gfCNCPoint3[20419] = {X 583.3023, Y 48.9046, Z -4.6667, A 0.000, B 0.000, C 0.000 }
gfCNCPoint3[20420] = {X 582.3585, Y 49.2242, Z -4.6667, A 0.000, B 0.000, C 0.000 }
gfCNCPoint3[20421] = {X 581.3666, Y 49.3191, Z -4.6667, A 0.000, B 0.000, C 0.000 }
gfCNCPoint3[20422] = {X 580.3794, Y 49.1842, Z -4.6667, A 0.000, B 0.000, C 0.000 }
gfCNCPoint3[20423] = {X 579.4493, Y 48.8268, Z -4.6667, A 0.000, B 0.000, C 0.000 }
gfCNCPoint3[20424] = {X 578.6259, Y 48.2657, Z -4.6667, A 0.000, B 0.000, C 0.000 }
gfCNCPoint3[20425] = {X 577.9529, Y 47.5309, Z -4.6667, A 0.000, B 0.000, C 0.000 }
gfCNCPoint3[20426] = {X 577.4662, Y 46.6615, Z -4.6667, A 0.000, B 0.000, C 0.000 }
gfCNCPoint3[20427] = {X 572.0189, Y 33.3415, Z -4.6667, A 0.000, B 0.000, C 0.000 }
gfCNCPoint3[20428] = {X 572.0192, Y 40.7711, Z -4.6667, A 0.000, B 0.000, C 0.000 }
gfCNCPoint3[20429] = {X 572.6574, Y 41.4420, Z -4.6667, A 0.000, B 0.000, C 0.000 }
gfCNCPoint3[20430] = {X 573.1380, Y 42.2334, Z -4.6667, A 0.000, B 0.000, C 0.000 }
gfCNCPoint3[20431] = {X 573.4389, Y 43.1090, Z -4.6667, A 0.000, B 0.000, C 0.000 }
gfCNCPoint3[20432] = {X 573.5463, Y 44.0287, Z -4.6667, A 0.000, B 0.000, C 0.000 }
gfCNCPoint3[20433] = {X 573.5464, Y 45.0000, Z -4.6667, A 0.000, B 0.000, C 0.000 }
gfCNCPoint3[20434] = {X 573.4381, Y 45.9613, Z -4.6667, A 0.000, B 0.000, C 0.000 }
gfCNCPoint3[20435] = {X 573.1186, Y 46.8744, Z -4.6667, A 0.000, B 0.000, C 0.000 }
gfCNCPoint3[20436] = {X 572.6039, Y 47.6935, Z -4.6667, A 0.000, B 0.000, C 0.000 }
gfCNCPoint3[20437] = {X 571.9199, Y 48.3775, Z -4.6667, A 0.000, B 0.000, C 0.000 }
gfCNCPoint3[20438] = {X 571.1008, Y 48.8922, Z -4.6667, A 0.000, B 0.000, C 0.000 }
gfCNCPoint3[20439] = {X 570.1877, Y 49.2117, Z -4.6667, A 0.000, B 0.000, C 0.000 }
gfCNCPoint3[20440] = {X 569.2264, Y 49.3200, Z -4.6667, A 0.000, B 0.000, C 0.000 }
gfCNCPoint3[20441] = {X 562.4443, Y 49.3200, Z -4.6667, A 0.000, B 0.000, C 0.000 }
gfCNCPoint3[20442] = {X 561.4830, Y 49.2117, Z -4.6667, A 0.000, B 0.000, C 0.000 }
gfCNCPoint3[20443] = {X 560.5699, Y 48.8922, Z -4.6667, A 0.000, B 0.000, C 0.000 }
gfCNCPoint3[20444] = {X 559.7508, Y 48.3775, Z -4.6667, A 0.000, B 0.000, C 0.000 }
gfCNCPoint3[20445] = {X 559.0668, Y 47.6935, Z -4.6667, A 0.000, B 0.000, C 0.000 }
gfCNCPoint3[20446] = {X 558.5521, Y 46.8744, Z -4.6667, A 0.000, B 0.000, C 0.000 }
gfCNCPoint3[20447] = {X 558.2326, Y 45.9613, Z -4.6667, A 0.000, B 0.000, C 0.000 }
gfCNCPoint3[20448] = {X 558.1243, Y 45.0000, Z -4.6667, A 0.000, B 0.000, C 0.000 }
gfCNCPoint3[20449] = {X 558.1243, Y 44.0647, Z -4.6667, A 0.000, B 0.000, C 0.000 }
gfCNCPoint3[20450] = {X 558.2284, Y 43.1360, Z -4.6667, A 0.000, B 0.000, C 0.000 }
gfCNCPoint3[20451] = {X 558.5283, Y 42.2510, Z -4.6667, A 0.000, B 0.000, C 0.000 }
gfCNCPoint3[20452] = {X 559.0102, Y 41.4503, Z -4.6667, A 0.000, B 0.000, C 0.000 }
gfCNCPoint3[20453] = {X 559.6518, Y 40.7709, Z -4.6667, A 0.000, B 0.000, C 0.000 }
gfCNCPoint3[20454] = {X 559.6518, Y 9.2302, Z -4.6667, A 0.000, B 0.000, C 0.000 }
gfCNCPoint3[20455] = {X 559.0134, Y 8.5592, Z -4.6667, A 0.000, B 0.000, C 0.000 }
gfCNCPoint3[20456] = {X 558.5327, Y 7.7676, Z -4.6667, A 0.000, B 0.000, C 0.000 }
gfCNCPoint3[20457] = {X 558.2318, Y 6.8917, Z -4.6667, A 0.000, B 0.000, C 0.000 }
gfCNCPoint3[20458] = {X 558.1245, Y 5.9718, Z -4.6667, A 0.000, B 0.000, C 0.000 }
gfCNCPoint3[20459] = {X 558.1243, Y 5.0000, Z -4.6667, A 0.000, B 0.000, C 0.000 }
gfCNCPoint3[20460] = {X 558.2326, Y 4.0387, Z -4.6667, A 0.000, B 0.000, C 0.000 }
gfCNCPoint3[20461] = {X 558.5521, Y 3.1256, Z -4.6667, A 0.000, B 0.000, C 0.000 }
gfCNCPoint3[20462] = {X 559.0668, Y 2.3065, Z -4.6667, A 0.000, B 0.000, C 0.000 }
gfCNCPoint3[20463] = {X 559.7508, Y 1.6225, Z -4.6667, A 0.000, B 0.000, C 0.000 }
gfCNCPoint3[20464] = {X 560.5699, Y 1.1078, Z -4.6667, A 0.000, B 0.000, C 0.000 }
gfCNCPoint3[20465] = {X 561.4830, Y 0.7883, Z -4.6667, A 0.000, B 0.000, C 0.000 }
gfCNCPoint3[20466] = {X 562.4443, Y 0.6800, Z -4.6667, A 0.000, B 0.000, C 0.000 }
gfCNCPoint3[20467] = {X 570.9376, Y 0.6800, Z -4.6667, A 0.000, B 0.000, C 0.000 }
gfCNCPoint3[20468] = {X 571.8988, Y 0.7883, Z -4.6667, A 0.000, B 0.000, C 0.000 }
gfCNCPoint3[20469] = {X 572.8119, Y 1.1078, Z -4.6667, A 0.000, B 0.000, C 0.000 }
gfCNCPoint3[20470] = {X 573.6310, Y 1.6225, Z -4.6667, A 0.000, B 0.000, C 0.000 }
gfCNCPoint3[20471] = {X 574.3151, Y 2.3065, Z -4.6667, A 0.000, B 0.000, C 0.000 }
gfCNCPoint3[20472] = {X 574.8297, Y 3.1256, Z -4.6667, A 0.000, B 0.000, C 0.000 }
gfCNCPoint3[20473] = {X 575.1492, Y 4.0387, Z -4.6667, A 0.000, B 0.000, C 0.000 }
gfCNCPoint3[20474] = {X 575.2576, Y 5.0000, Z -4.6667, A 0.000, B 0.000, C 0.000 }
gfCNCPoint3[20475] = {X 575.2576, Y 5.9342, Z -4.6667, A 0.000, B 0.000, C 0.000 }
gfCNCPoint3[20476] = {X 575.1835, Y 6.7305, Z -4.6667, A 0.000, B 0.000, C 0.000 }
gfCNCPoint3[20477] = {X 574.9639, Y 7.4995, Z -4.6667, A 0.000, B 0.000, C 0.000 }
gfCNCPoint3[20478] = {X 574.6064, Y 8.2149, Z -4.6667, A 0.000, B 0.000, C 0.000 }
gfCNCPoint3[20479] = {X 581.1910, Y 24.3698, Z -4.6667, A 0.000, B 0.000, C 0.000 }
gfCNCPoint3[20480] = {X 587.8458, Y 8.0941, Z -4.6667, A 0.000, B 0.000, C 0.000 }
gfCNCPoint3[20481] = {X 587.5317, Y 7.4230, Z -4.6667, A 0.000, B 0.000, C 0.000 }
gfCNCPoint3[20482] = {X 587.3369, Y 6.7082, Z -4.6667, A 0.000, B 0.000, C 0.000 }
gfCNCPoint3[20483] = {X 587.2671, Y 5.9705, Z -4.6667, A 0.000, B 0.000, C 0.000 }
gfCNCPoint3[20484] = {X 587.2670, Y 5.0000, Z -4.6667, A 0.000, B 0.000, C 0.000 }
gfCNCPoint3[20485] = {X 587.3753, Y 4.0387, Z -4.6667, A 0.000, B 0.000, C 0.000 }
gfCNCPoint3[20486] = {X 587.6948, Y 3.1256, Z -4.6667, A 0.000, B 0.000, C 0.000 }
gfCNCPoint3[20487] = {X 588.2094, Y 2.3065, Z -4.6667, A 0.000, B 0.000, C 0.000 }
gfCNCPoint3[20488] = {X 588.8935, Y 1.6225, Z -4.6667, A 0.000, B 0.000, C 0.000 }
gfCNCPoint3[20489] = {X 589.7126, Y 1.1078, Z -4.6667, A 0.000, B 0.000, C 0.000 }
gfCNCPoint3[20490] = {X 590.6257, Y 0.7883, Z -4.6667, A 0.000, B 0.000, C 0.000 }
gfCNCPoint3[20491] = {X 591.5870, Y 0.6800, Z -4.6667, A 0.000, B 0.000, C 0.000 }
gfCNCPoint3[20492] = {X 600.0000, Y 0.6800, Z -4.6667, A 0.000, B 0.000, C 0.000 }
gfCNCPoint3[20493] = {X 600.8562, Y 0.7657, Z -4.6667, A 0.000, B 0.000, C 0.000 }
gfCNCPoint3[20494] = {X 601.6783, Y 1.0194, Z -4.6667, A 0.000, B 0.000, C 0.000 }
gfCNCPoint3[20495] = {X 602.4340, Y 1.4309, Z -4.6667, A 0.000, B 0.000, C 0.000 }
gfCNCPoint3[20496] = {X 603.0930, Y 1.9841, Z -4.6667, A 0.000, B 0.000, C 0.000 }
gfCNCPoint3[20497] = {X 603.6294, Y 2.6569, Z -4.6667, A 0.000, B 0.000, C 0.000 }
gfCNCPoint3[20498] = {X 603.6634, Y 2.7104, Z -4.6667, A 0.000, B 0.000, C 0.000 }
gfCNCPoint3[20499] = {X 603.6966, Y 2.7644, Z -4.6667, A 0.000, B 0.000, C 0.000 }
gfCNCPoint3[20500] = {X 608.0000, Y 9.8803, Z -4.6667, A 0.000, B 0.000, C 0.000 }
gfCNCPoint3[20501] = {X 608.0000, Y 9.8803, Z -1.6667, A 0.000, B 0.000, C 0.000 }
gfCNCPoint3[20502] = {X 608.0000, Y 9.8803, Z 11.0000, A 0.000, B 0.000, C 0.000 }
gfCNCPoint3[20503] = {X -7.6966, Y 16.7865, Z 11.0000, A 0.000, B 0.000, C 0.000 }
gfCNCPoint3[20504] = {X -7.6966, Y 16.7865, Z -1.6667, A 0.000, B 0.000, C 0.000 }
gfCNCPoint3[20505] = {X -7.6966, Y 16.7865, Z -4.6667, A 0.000, B 0.000, C 0.000 }
gfCNCPoint3[20506] = {X -4.6244, Y 16.7865, Z -4.6667, A 0.000, B 0.000, C 0.000 }
gfCNCPoint3[20507] = {X -3.6966, Y 12.8956, Z -4.6667, A 0.000, B 0.000, C 0.000 }
gfCNCPoint3[20508] = {X -3.6291, Y 12.6465, Z -4.6667, A 0.000, B 0.000, C 0.000 }
gfCNCPoint3[20509] = {X -3.5466, Y 12.4020, Z -4.6667, A 0.000, B 0.000, C 0.000 }
gfCNCPoint3[20510] = {X -3.1001, Y 11.5272, Z -4.6667, A 0.000, B 0.000, C 0.000 }
gfCNCPoint3[20511] = {X -2.4643, Y 10.7786, Z -4.6667, A 0.000, B 0.000, C 0.000 }
gfCNCPoint3[20512] = {X -1.6733, Y 10.1963, Z -4.6667, A 0.000, B 0.000, C 0.000 }
gfCNCPoint3[20513] = {X -1.0760, Y 9.8556, Z -4.6667, A 0.000, B 0.000, C 0.000 }
gfCNCPoint3[20514] = {X -0.1979, Y 9.4786, Z -4.6667, A 0.000, B 0.000, C 0.000 }
gfCNCPoint3[20515] = {X 0.7423, Y 9.3079, Z -4.6667, A 0.000, B 0.000, C 0.000 }
gfCNCPoint3[20516] = {X 1.6969, Y 9.3520, Z -4.6667, A 0.000, B 0.000, C 0.000 }
gfCNCPoint3[20517] = {X 2.6173, Y 9.6089, Z -4.6667, A 0.000, B 0.000, C 0.000 }
gfCNCPoint3[20518] = {X 3.4039, Y 9.2325, Z -4.6667, A 0.000, B 0.000, C 0.000 }
gfCNCPoint3[20519] = {X 4.2182, Y 8.9206, Z -4.6667, A 0.000, B 0.000, C 0.000 }
gfCNCPoint3[20520] = {X 6.1238, Y 8.2532, Z -4.6667, A 0.000, B 0.000, C 0.000 }
gfCNCPoint3[20521] = {X 8.0799, Y 7.7526, Z -4.6667, A 0.000, B 0.000, C 0.000 }
gfCNCPoint3[20522] = {X 10.0718, Y 7.4226, Z -4.6667, A 0.000, B 0.000, C 0.000 }
gfCNCPoint3[20523] = {X 12.0848, Y 7.2658, Z -4.6667, A 0.000, B 0.000, C 0.000 }
gfCNCPoint3[20524] = {X 14.1038, Y 7.2832, Z -4.6667, A 0.000, B 0.000, C 0.000 }
gfCNCPoint3[20525] = {X 16.1138, Y 7.4747, Z -4.6667, A 0.000, B 0.000, C 0.000 }
gfCNCPoint3[20526] = {X 17.9288, Y 7.8067, Z -4.6667, A 0.000, B 0.000, C 0.000 }
gfCNCPoint3[20527] = {X 19.6983, Y 8.3293, Z -4.6667, A 0.000, B 0.000, C 0.000 }
gfCNCPoint3[20528] = {X 21.4023, Y 9.0367, Z -4.6667, A 0.000, B 0.000, C 0.000 }
gfCNCPoint3[20529] = {X 23.0218, Y 9.9207, Z -4.6667, A 0.000, B 0.000, C 0.000 }
gfCNCPoint3[20530] = {X 24.5384, Y 10.9716, Z -4.6667, A 0.000, B 0.000, C 0.000 }
gfCNCPoint3[20531] = {X 25.6169, Y 11.9146, Z -4.6667, A 0.000, B 0.000, C 0.000 }
gfCNCPoint3[20532] = {X 26.5844, Y 12.9712, Z -4.6667, A 0.000, B 0.000, C 0.000 }
gfCNCPoint3[20533] = {X 27.4289, Y 14.1285, Z -4.6667, A 0.000, B 0.000, C 0.000 }
gfCNCPoint3[20534] = {X 28.1401, Y 15.3722, Z -4.6667, A 0.000, B 0.000, C 0.000 }
gfCNCPoint3[20535] = {X 28.7091, Y 16.6870, Z -4.6667, A 0.000, B 0.000, C 0.000 }
gfCNCPoint3[20536] = {X 29.1816, Y 18.3343, Z -4.6667, A 0.000, B 0.000, C 0.000 }
gfCNCPoint3[20537] = {X 29.4619, Y 20.0250, Z -4.6667, A 0.000, B 0.000, C 0.000 }
gfCNCPoint3[20538] = {X 29.5464, Y 21.7367, Z -4.6667, A 0.000, B 0.000, C 0.000 }
gfCNCPoint3[20539] = {X 29.4338, Y 23.4467, Z -4.6667, A 0.000, B 0.000, C 0.000 }
gfCNCPoint3[20540] = {X 29.1258, Y 25.1326, Z -4.6667, A 0.000, B 0.000, C 0.000 }
gfCNCPoint3[20541] = {X 28.6966, Y 26.5422, Z -4.6667, A 0.000, B 0.000, C 0.000 }
gfCNCPoint3[20542] = {X 28.0924, Y 27.8862, Z -4.6667, A 0.000, B 0.000, C 0.000 }
gfCNCPoint3[20543] = {X 27.3227, Y 29.1428, Z -4.6667, A 0.000, B 0.000, C 0.000 }
gfCNCPoint3[20544] = {X 26.4001, Y 30.2918, Z -4.6667, A 0.000, B 0.000, C 0.000 }
gfCNCPoint3[20545] = {X 25.3394, Y 31.3146, Z -4.6667, A 0.000, B 0.000, C 0.000 }
gfCNCPoint3[20546] = {X 25.2268, Y 31.4090, Z -4.6667, A 0.000, B 0.000, C 0.000 }
gfCNCPoint3[20547] = {X 25.1130, Y 31.5020, Z -4.6667, A 0.000, B 0.000, C 0.000 }
gfCNCPoint3[20548] = {X 25.9470, Y 31.8267, Z -4.6667, A 0.000, B 0.000, C 0.000 }
gfCNCPoint3[20549] = {X 26.6943, Y 32.3192, Z -4.6667, A 0.000, B 0.000, C 0.000 }
gfCNCPoint3[20550] = {X 27.3216, Y 32.9577, Z -4.6667, A 0.000, B 0.000, C 0.000 }
gfCNCPoint3[20551] = {X 27.8009, Y 33.7136, Z -4.6667, A 0.000, B 0.000, C 0.000 }
gfCNCPoint3[20552] = {X 30.8380, Y 39.9879, Z -4.6667, A 0.000, B 0.000, C 0.000 }
gfCNCPoint3[20553] = {X 31.1526, Y 40.8802, Z -4.6667, A 0.000, B 0.000, C 0.000 }
gfCNCPoint3[20554] = {X 31.2615, Y 41.8200, Z -4.6667, A 0.000, B 0.000, C 0.000 }
gfCNCPoint3[20555] = {X 31.1593, Y 42.7606, Z -4.6667, A 0.000, B 0.000, C 0.000 }
gfCNCPoint3[20556] = {X 30.8511, Y 43.6551, Z -4.6667, A 0.000, B 0.000, C 0.000 }
gfCNCPoint3[20557] = {X 30.3522, Y 44.4590, Z -4.6667, A 0.000, B 0.000, C 0.000 }
gfCNCPoint3[20558] = {X 29.6874, Y 45.1323, Z -4.6667, A 0.000, B 0.000, C 0.000 }
gfCNCPoint3[20559] = {X 29.1513, Y 45.5657, Z -4.6667, A 0.000, B 0.000, C 0.000 }
gfCNCPoint3[20560] = {X 28.4540, Y 46.0238, Z -4.6667, A 0.000, B 0.000, C 0.000 }
gfCNCPoint3[20561] = {X 27.6807, Y 46.3369, Z -4.6667, A 0.000, B 0.000, C 0.000 }
gfCNCPoint3[20562] = {X 26.8611, Y 46.4931, Z -4.6667, A 0.000, B 0.000, C 0.000 }
gfCNCPoint3[20563] = {X 26.0268, Y 46.4863, Z -4.6667, A 0.000, B 0.000, C 0.000 }
gfCNCPoint3[20564] = {X 25.2099, Y 46.3169, Z -4.6667, A 0.000, B 0.000, C 0.000 }
gfCNCPoint3[20565] = {X 23.4056, Y 47.2718, Z -4.6667, A 0.000, B 0.000, C 0.000 }
gfCNCPoint3[20566] = {X 21.5389, Y 48.0979, Z -4.6667, A 0.000, B 0.000, C 0.000 }
gfCNCPoint3[20567] = {X 19.6188, Y 48.7912, Z -4.6667, A 0.000, B 0.000, C 0.000 }
gfCNCPoint3[20568] = {X 17.6857, Y 49.3364, Z -4.6667, A 0.000, B 0.000, C 0.000 }
gfCNCPoint3[20569] = {X 15.7120, Y 49.7085, Z -4.6667, A 0.000, B 0.000, C 0.000 }
gfCNCPoint3[20570] = {X 13.7132, Y 49.9048, Z -4.6667, A 0.000, B 0.000, C 0.000 }
gfCNCPoint3[20571] = {X 11.7048, Y 49.9236, Z -4.6667, A 0.000, B 0.000, C 0.000 }
gfCNCPoint3[20572] = {X 9.7026, Y 49.7647, Z -4.6667, A 0.000, B 0.000, C 0.000 }
gfCNCPoint3[20573] = {X 7.7223, Y 49.4296, Z -4.6667, A 0.000, B 0.000, C 0.000 }
gfCNCPoint3[20574] = {X 5.8294, Y 48.9112, Z -4.6667, A 0.000, B 0.000, C 0.000 }
gfCNCPoint3[20575] = {X 4.0107, Y 48.1734, Z -4.6667, A 0.000, B 0.000, C 0.000 }
gfCNCPoint3[20576] = {X 2.2918, Y 47.2262, Z -4.6667, A 0.000, B 0.000, C 0.000 }
gfCNCPoint3[20577] = {X 0.6965, Y 46.0830, Z -4.6667, A 0.000, B 0.000, C 0.000 }
gfCNCPoint3[20578] = {X -0.4291, Y 45.0714, Z -4.6667, A 0.000, B 0.000, C 0.000 }
gfCNCPoint3[20579] = {X -1.4287, Y 43.9351, Z -4.6667, A 0.000, B 0.000, C 0.000 }
gfCNCPoint3[20580] = {X -2.2886, Y 42.6898, Z -4.6667, A 0.000, B 0.000, C 0.000 }
gfCNCPoint3[20581] = {X -2.9970, Y 41.3524, Z -4.6667, A 0.000, B 0.000, C 0.000 }
gfCNCPoint3[20582] = {X -3.5443, Y 39.9415, Z -4.6667, A 0.000, B 0.000, C 0.000 }
gfCNCPoint3[20583] = {X -3.6230, Y 39.6879, Z -4.6667, A 0.000, B 0.000, C 0.000 }
gfCNCPoint3[20584] = {X -3.6966, Y 39.4327, Z -4.6667, A 0.000, B 0.000, C 0.000 }
gfCNCPoint3[20585] = {X -4.7647, Y 35.5779, Z -4.6667, A 0.000, B 0.000, C 0.000 }
gfCNCPoint3[20586] = {X -8.0037, Y 35.6277, Z -4.6667, A 0.000, B 0.000, C 0.000 }
gfCNCPoint3[20587] = {X -8.0037, Y 35.6277, Z -1.6667, A 0.000, B 0.000, C 0.000 }
gfCNCPoint3[20588] = {X -8.0037, Y 35.6277, Z 11.0000, A 0.000, B 0.000, C 0.000 }
gfCNCPoint3[20589] = {X -7.6966, Y 17.3015, Z 11.0000, A 0.000, B 0.000, C 0.000 }
gfCNCPoint3[20590] = {X -7.6966, Y 17.3015, Z -1.6667, A 0.000, B 0.000, C 0.000 }
gfCNCPoint3[20591] = {X -7.6966, Y 17.3015, Z -4.6667, A 0.000, B 0.000, C 0.000 }
gfCNCPoint3[20592] = {X -4.2191, Y 17.3015, Z -4.6667, A 0.000, B 0.000, C 0.000 }
gfCNCPoint3[20593] = {X -3.6966, Y 13.3357, Z -4.6667, A 0.000, B 0.000, C 0.000 }
gfCNCPoint3[20594] = {X -3.6096, Y 12.8765, Z -4.6667, A 0.000, B 0.000, C 0.000 }
gfCNCPoint3[20595] = {X -3.4716, Y 12.4299, Z -4.6667, A 0.000, B 0.000, C 0.000 }
gfCNCPoint3[20596] = {X -3.0335, Y 11.5715, Z -4.6667, A 0.000, B 0.000, C 0.000 }
gfCNCPoint3[20597] = {X -2.4097, Y 10.8371, Z -4.6667, A 0.000, B 0.000, C 0.000 }
gfCNCPoint3[20598] = {X -1.6337, Y 10.2658, Z -4.6667, A 0.000, B 0.000, C 0.000 }
gfCNCPoint3[20599] = {X -1.0364, Y 9.9251, Z -4.6667, A 0.000, B 0.000, C 0.000 }
gfCNCPoint3[20600] = {X -0.1659, Y 9.5525, Z -4.6667, A 0.000, B 0.000, C 0.000 }
gfCNCPoint3[20601] = {X 0.7662, Y 9.3865, Z -4.6667, A 0.000, B 0.000, C 0.000 }
gfCNCPoint3[20602] = {X 1.7117, Y 9.4356, Z -4.6667, A 0.000, B 0.000, C 0.000 }
gfCNCPoint3[20603] = {X 2.6217, Y 9.6971, Z -4.6667, A 0.000, B 0.000, C 0.000 }
gfCNCPoint3[20604] = {X 3.4193, Y 9.3129, Z -4.6667, A 0.000, B 0.000, C 0.000 }
gfCNCPoint3[20605] = {X 4.2459, Y 8.9957, Z -4.6667, A 0.000, B 0.000, C 0.000 }
gfCNCPoint3[20606] = {X 6.1453, Y 8.3302, Z -4.6667, A 0.000, B 0.000, C 0.000 }
gfCNCPoint3[20607] = {X 8.0950, Y 7.8311, Z -4.6667, A 0.000, B 0.000, C 0.000 }
gfCNCPoint3[20608] = {X 10.0806, Y 7.5022, Z -4.6667, A 0.000, B 0.000, C 0.000 }
gfCNCPoint3[20609] = {X 12.0871, Y 7.3458, Z -4.6667, A 0.000, B 0.000, C 0.000 }
gfCNCPoint3[20610] = {X 14.0997, Y 7.3631, Z -4.6667, A 0.000, B 0.000, C 0.000 }
gfCNCPoint3[20611] = {X 16.1032, Y 7.5540, Z -4.6667, A 0.000, B 0.000, C 0.000 }
gfCNCPoint3[20612] = {X 17.9099, Y 7.8845, Z -4.6667, A 0.000, B 0.000, C 0.000 }
gfCNCPoint3[20613] = {X 19.6713, Y 8.4047, Z -4.6667, A 0.000, B 0.000, C 0.000 }
gfCNCPoint3[20614] = {X 21.3676, Y 9.1088, Z -4.6667, A 0.000, B 0.000, C 0.000 }
gfCNCPoint3[20615] = {X 22.9797, Y 9.9888, Z -4.6667, A 0.000, B 0.000, C 0.000 }
gfCNCPoint3[20616] = {X 24.4894, Y 11.0348, Z -4.6667, A 0.000, B 0.000, C 0.000 }
gfCNCPoint3[20617] = {X 25.5612, Y 11.9720, Z -4.6667, A 0.000, B 0.000, C 0.000 }
gfCNCPoint3[20618] = {X 26.5226, Y 13.0220, Z -4.6667, A 0.000, B 0.000, C 0.000 }
gfCNCPoint3[20619] = {X 27.3618, Y 14.1721, Z -4.6667, A 0.000, B 0.000, C 0.000 }
gfCNCPoint3[20620] = {X 28.0685, Y 15.4081, Z -4.6667, A 0.000, B 0.000, C 0.000 }
gfCNCPoint3[20621] = {X 28.6341, Y 16.7146, Z -4.6667, A 0.000, B 0.000, C 0.000 }
gfCNCPoint3[20622] = {X 29.1038, Y 18.3530, Z -4.6667, A 0.000, B 0.000, C 0.000 }
gfCNCPoint3[20623] = {X 29.3825, Y 20.0344, Z -4.6667, A 0.000, B 0.000, C 0.000 }
gfCNCPoint3[20624] = {X 29.4664, Y 21.7367, Z -4.6667, A 0.000, B 0.000, C 0.000 }
gfCNCPoint3[20625] = {X 29.3544, Y 23.4373, Z -4.6667, A 0.000, B 0.000, C 0.000 }
gfCNCPoint3[20626] = {X 29.0480, Y 25.1139, Z -4.6667, A 0.000, B 0.000, C 0.000 }
gfCNCPoint3[20627] = {X 28.6218, Y 26.5139, Z -4.6667, A 0.000, B 0.000, C 0.000 }
gfCNCPoint3[20628] = {X 28.0217, Y 27.8487, Z -4.6667, A 0.000, B 0.000, C 0.000 }
gfCNCPoint3[20629] = {X 27.2574, Y 29.0967, Z -4.6667, A 0.000, B 0.000, C 0.000 }
gfCNCPoint3[20630] = {X 26.3411, Y 30.2378, Z -4.6667, A 0.000, B 0.000, C 0.000 }
gfCNCPoint3[20631] = {X 25.2877, Y 31.2536, Z -4.6667, A 0.000, B 0.000, C 0.000 }
gfCNCPoint3[20632] = {X 25.1135, Y 31.3986, Z -4.6667, A 0.000, B 0.000, C 0.000 }
gfCNCPoint3[20633] = {X 24.9364, Y 31.5401, Z -4.6667, A 0.000, B 0.000, C 0.000 }
gfCNCPoint3[20634] = {X 25.8026, Y 31.8441, Z -4.6667, A 0.000, B 0.000, C 0.000 }
gfCNCPoint3[20635] = {X 26.5811, Y 32.3307, Z -4.6667, A 0.000, B 0.000, C 0.000 }
gfCNCPoint3[20636] = {X 27.2339, Y 32.9761, Z -4.6667, A 0.000, B 0.000, C 0.000 }
gfCNCPoint3[20637] = {X 27.7292, Y 33.7491, Z -4.6667, A 0.000, B 0.000, C 0.000 }
gfCNCPoint3[20638] = {X 30.7660, Y 40.0227, Z -4.6667, A 0.000, B 0.000, C 0.000 }
gfCNCPoint3[20639] = {X 31.0747, Y 40.8982, Z -4.6667, A 0.000, B 0.000, C 0.000 }
gfCNCPoint3[20640] = {X 31.1815, Y 41.8203, Z -4.6667, A 0.000, B 0.000, C 0.000 }
gfCNCPoint3[20641] = {X 31.0813, Y 42.7431, Z -4.6667, A 0.000, B 0.000, C 0.000 }
gfCNCPoint3[20642] = {X 30.7789, Y 43.6208, Z -4.6667, A 0.000, B 0.000, C 0.000 }
gfCNCPoint3[20643] = {X 30.2893, Y 44.4095, Z -4.6667, A 0.000, B 0.000, C 0.000 }
gfCNCPoint3[20644] = {X 29.6371, Y 45.0700, Z -4.6667, A 0.000, B 0.000, C 0.000 }
gfCNCPoint3[20645] = {X 29.1010, Y 45.5035, Z -4.6667, A 0.000, B 0.000, C 0.000 }
gfCNCPoint3[20646] = {X 28.4106, Y 45.9562, Z -4.6667, A 0.000, B 0.000, C 0.000 }
gfCNCPoint3[20647] = {X 27.6446, Y 46.2641, Z -4.6667, A 0.000, B 0.000, C 0.000 }
gfCNCPoint3[20648] = {X 26.8330, Y 46.4153, Z -4.6667, A 0.000, B 0.000, C 0.000 }
gfCNCPoint3[20649] = {X 26.0076, Y 46.4037, Z -4.6667, A 0.000, B 0.000, C 0.000 }
gfCNCPoint3[20650] = {X 25.2005, Y 46.2300, Z -4.6667, A 0.000, B 0.000, C 0.000 }
gfCNCPoint3[20651] = {X 23.3917, Y 47.1896, Z -4.6667, A 0.000, B 0.000, C 0.000 }
gfCNCPoint3[20652] = {X 21.5197, Y 48.0194, Z -4.6667, A 0.000, B 0.000, C 0.000 }
gfCNCPoint3[20653] = {X 19.5939, Y 48.7152, Z -4.6667, A 0.000, B 0.000, C 0.000 }
gfCNCPoint3[20654] = {X 19.4378, Y 48.7674, Z -4.6667, A 0.000, B 0.000, C 0.000 }
gfCNCPoint3[20655] = {X 17.5342, Y 49.2904, Z -4.6667, A 0.000, B 0.000, C 0.000 }
gfCNCPoint3[20656] = {X 15.5923, Y 49.6454, Z -4.6667, A 0.000, B 0.000, C 0.000 }
gfCNCPoint3[20657] = {X 13.6268, Y 49.8298, Z -4.6667, A 0.000, B 0.000, C 0.000 }
gfCNCPoint3[20658] = {X 11.6528, Y 49.8420, Z -4.6667, A 0.000, B 0.000, C 0.000 }
gfCNCPoint3[20659] = {X 9.6852, Y 49.6822, Z -4.6667, A 0.000, B 0.000, C 0.000 }
gfCNCPoint3[20660] = {X 7.7390, Y 49.3513, Z -4.6667, A 0.000, B 0.000, C 0.000 }
gfCNCPoint3[20661] = {X 5.8551, Y 48.8355, Z -4.6667, A 0.000, B 0.000, C 0.000 }
gfCNCPoint3[20662] = {X 4.0451, Y 48.1011, Z -4.6667, A 0.000, B 0.000, C 0.000 }
gfCNCPoint3[20663] = {X 2.3343, Y 47.1585, Z -4.6667, A 0.000, B 0.000, C 0.000 }
gfCNCPoint3[20664] = {X 0.7466, Y 46.0207, Z -4.6667, A 0.000, B 0.000, C 0.000 }
gfCNCPoint3[20665] = {X -0.3720, Y 45.0153, Z -4.6667, A 0.000, B 0.000, C 0.000 }
gfCNCPoint3[20666] = {X -1.3655, Y 43.8860, Z -4.6667, A 0.000, B 0.000, C 0.000 }
gfCNCPoint3[20667] = {X -2.2201, Y 42.6483, Z -4.6667, A 0.000, B 0.000, C 0.000 }
gfCNCPoint3[20668] = {X -2.9242, Y 41.3192, Z -4.6667, A 0.000, B 0.000, C 0.000 }
gfCNCPoint3[20669] = {X -3.4681, Y 39.9170, Z -4.6667, A 0.000, B 0.000, C 0.000 }
gfCNCPoint3[20670] = {X -3.5888, Y 39.5202, Z -4.6667, A 0.000, B 0.000, C 0.000 }
gfCNCPoint3[20671] = {X -3.6966, Y 39.1199, Z -4.6667, A 0.000, B 0.000, C 0.000 }
gfCNCPoint3[20672] = {X -4.6739, Y 35.2411, Z -4.6667, A 0.000, B 0.000, C 0.000 }
gfCNCPoint3[20673] = {X -8.0055, Y 35.2186, Z -4.6667, A 0.000, B 0.000, C 0.000 }
gfCNCPoint3[20674] = {X -8.0055, Y 35.2186, Z -1.6667, A 0.000, B 0.000, C 0.000 }
gfCNCPoint3[20675] = {X -8.0055, Y 35.2186, Z 11.0000, A 0.000, B 0.000, C 0.000 }
gfCNCPoint3[20676] = {X -7.9982, Y 34.8106, Z 11.0000, A 0.000, B 0.000, C 0.000 }
gfCNCPoint3[20677] = {X -7.9982, Y 34.8106, Z -1.6667, A 0.000, B 0.000, C 0.000 }
gfCNCPoint3[20678] = {X -7.9982, Y 34.8106, Z -4.6667, A 0.000, B 0.000, C 0.000 }
gfCNCPoint3[20679] = {X -4.8500, Y 34.9014, Z -4.6667, A 0.000, B 0.000, C 0.000 }
gfCNCPoint3[20680] = {X -3.6966, Y 31.0713, Z -4.6667, A 0.000, B 0.000, C 0.000 }
gfCNCPoint3[20681] = {X -3.6590, Y 30.9485, Z -4.6667, A 0.000, B 0.000, C 0.000 }
gfCNCPoint3[20682] = {X -3.6204, Y 30.8260, Z -4.6667, A 0.000, B 0.000, C 0.000 }
gfCNCPoint3[20683] = {X -3.4453, Y 30.3119, Z -4.6667, A 0.000, B 0.000, C 0.000 }
gfCNCPoint3[20684] = {X -3.2516, Y 29.8045, Z -4.6667, A 0.000, B 0.000, C 0.000 }
gfCNCPoint3[20685] = {X -2.6170, Y 28.4651, Z -4.6667, A 0.000, B 0.000, C 0.000 }
gfCNCPoint3[20686] = {X -1.8053, Y 27.2250, Z -4.6667, A 0.000, B 0.000, C 0.000 }
gfCNCPoint3[20687] = {X -0.8319, Y 26.1073, Z -4.6667, A 0.000, B 0.000, C 0.000 }
gfCNCPoint3[20688] = {X 0.2851, Y 25.1331, Z -4.6667, A 0.000, B 0.000, C 0.000 }
gfCNCPoint3[20689] = {X 1.5247, Y 24.3206, Z -4.6667, A 0.000, B 0.000, C 0.000 }
gfCNCPoint3[20690] = {X 0.7362, Y 23.9298, Z -4.6667, A 0.000, B 0.000, C 0.000 }
gfCNCPoint3[20691] = {X 0.0433, Y 23.3873, Z -4.6667, A 0.000, B 0.000, C 0.000 }
gfCNCPoint3[20692] = {X -0.5253, Y 22.7156, Z -4.6667, A 0.000, B 0.000, C 0.000 }
gfCNCPoint3[20693] = {X -0.9460, Y 21.9427, Z -4.6667, A 0.000, B 0.000, C 0.000 }
gfCNCPoint3[20694] = {X -3.6216, Y 15.3841, Z -4.6667, A 0.000, B 0.000, C 0.000 }
gfCNCPoint3[20695] = {X -3.6606, Y 15.2748, Z -4.6667, A 0.000, B 0.000, C 0.000 }
gfCNCPoint3[20696] = {X -3.6966, Y 15.1645, Z -4.6667, A 0.000, B 0.000, C 0.000 }
gfCNCPoint3[20697] = {X -4.8867, Y 11.3456, Z -4.6667, A 0.000, B 0.000, C 0.000 }
gfCNCPoint3[20698] = {X -7.6966, Y 11.3456, Z -4.6667, A 0.000, B 0.000, C 0.000 }
gfCNCPoint3[20699] = {X -7.6966, Y 11.3456, Z -1.6667, A 0.000, B 0.000, C 0.000 }
gfCNCPoint3[20700] = {X -7.6966, Y 11.3456, Z 11.0000, A 0.000, B 0.000, C 0.000 }
gfCNCPoint3[20701] = {X -8.0052, Y 35.1799, Z 11.0000, A 0.000, B 0.000, C 0.000 }
gfCNCPoint3[20702] = {X -8.0052, Y 35.1799, Z -1.6667, A 0.000, B 0.000, C 0.000 }
gfCNCPoint3[20703] = {X -8.0052, Y 35.1799, Z -4.6667, A 0.000, B 0.000, C 0.000 }
gfCNCPoint3[20704] = {X -4.7785, Y 35.2084, Z -4.6667, A 0.000, B 0.000, C 0.000 }
gfCNCPoint3[20705] = {X -3.6966, Y 31.3575, Z -4.6667, A 0.000, B 0.000, C 0.000 }
gfCNCPoint3[20706] = {X -3.6227, Y 31.1033, Z -4.6667, A 0.000, B 0.000, C 0.000 }
gfCNCPoint3[20707] = {X -3.5442, Y 30.8504, Z -4.6667, A 0.000, B 0.000, C 0.000 }
gfCNCPoint3[20708] = {X -3.3700, Y 30.3389, Z -4.6667, A 0.000, B 0.000, C 0.000 }
gfCNCPoint3[20709] = {X -3.1772, Y 29.8341, Z -4.6667, A 0.000, B 0.000, C 0.000 }
gfCNCPoint3[20710] = {X -2.5634, Y 28.5332, Z -4.6667, A 0.000, B 0.000, C 0.000 }
gfCNCPoint3[20711] = {X -1.7812, Y 27.3260, Z -4.6667, A 0.000, B 0.000, C 0.000 }
gfCNCPoint3[20712] = {X -0.8449, Y 26.2341, Z -4.6667, A 0.000, B 0.000, C 0.000 }
gfCNCPoint3[20713] = {X 0.2290, Y 25.2770, Z -4.6667, A 0.000, B 0.000, C 0.000 }
gfCNCPoint3[20714] = {X 1.4210, Y 24.4720, Z -4.6667, A 0.000, B 0.000, C 0.000 }
gfCNCPoint3[20715] = {X 1.5699, Y 24.3870, Z -4.6667, A 0.000, B 0.000, C 0.000 }
gfCNCPoint3[20716] = {X 1.7200, Y 24.3043, Z -4.6667, A 0.000, B 0.000, C 0.000 }
gfCNCPoint3[20717] = {X 0.8925, Y 23.9312, Z -4.6667, A 0.000, B 0.000, C 0.000 }
gfCNCPoint3[20718] = {X 0.1633, Y 23.3904, Z -4.6667, A 0.000, B 0.000, C 0.000 }
gfCNCPoint3[20719] = {X -0.4340, Y 22.7069, Z -4.6667, A 0.000, B 0.000, C 0.000 }
gfCNCPoint3[20720] = {X -0.8722, Y 21.9118, Z -4.6667, A 0.000, B 0.000, C 0.000 }
gfCNCPoint3[20721] = {X -3.5466, Y 15.3562, Z -4.6667, A 0.000, B 0.000, C 0.000 }
gfCNCPoint3[20722] = {X -3.6291, Y 15.1117, Z -4.6667, A 0.000, B 0.000, C 0.000 }
gfCNCPoint3[20723] = {X -3.6966, Y 14.8626, Z -4.6667, A 0.000, B 0.000, C 0.000 }
gfCNCPoint3[20724] = {X -4.6244, Y 10.9717, Z -4.6667, A 0.000, B 0.000, C 0.000 }
gfCNCPoint3[20725] = {X -7.6966, Y 10.9717, Z -4.6667, A 0.000, B 0.000, C 0.000 }
gfCNCPoint3[20726] = {X -7.6966, Y 10.9717, Z -1.6667, A 0.000, B 0.000, C 0.000 }
gfCNCPoint3[20727] = {X -7.6966, Y 10.9717, Z 11.0000, A 0.000, B 0.000, C 0.000 }
gfCNCPoint3[20728] = {X -8.0044, Y 35.5781, Z 11.0000, A 0.000, B 0.000, C 0.000 }
gfCNCPoint3[20729] = {X -8.0044, Y 35.5781, Z -1.6667, A 0.000, B 0.000, C 0.000 }
gfCNCPoint3[20730] = {X -8.0044, Y 35.5781, Z -4.6667, A 0.000, B 0.000, C 0.000 }
gfCNCPoint3[20731] = {X -4.7007, Y 35.5362, Z -4.6667, A 0.000, B 0.000, C 0.000 }
gfCNCPoint3[20732] = {X -3.6966, Y 31.6643, Z -4.6667, A 0.000, B 0.000, C 0.000 }
gfCNCPoint3[20733] = {X -3.5878, Y 31.2679, Z -4.6667, A 0.000, B 0.000, C 0.000 }
gfCNCPoint3[20734] = {X -3.4680, Y 30.8748, Z -4.6667, A 0.000, B 0.000, C 0.000 }
gfCNCPoint3[20735] = {X -3.2947, Y 30.3659, Z -4.6667, A 0.000, B 0.000, C 0.000 }
gfCNCPoint3[20736] = {X -3.1029, Y 29.8637, Z -4.6667, A 0.000, B 0.000, C 0.000 }
gfCNCPoint3[20737] = {X -2.4936, Y 28.5724, Z -4.6667, A 0.000, B 0.000, C 0.000 }
gfCNCPoint3[20738] = {X -1.7173, Y 27.3741, Z -4.6667, A 0.000, B 0.000, C 0.000 }
gfCNCPoint3[20739] = {X -0.7879, Y 26.2902, Z -4.6667, A 0.000, B 0.000, C 0.000 }
gfCNCPoint3[20740] = {X 0.2780, Y 25.3402, Z -4.6667, A 0.000, B 0.000, C 0.000 }
gfCNCPoint3[20741] = {X 1.4613, Y 24.5411, Z -4.6667, A 0.000, B 0.000, C 0.000 }
gfCNCPoint3[20742] = {X 1.6938, Y 24.4097, Z -4.6667, A 0.000, B 0.000, C 0.000 }
gfCNCPoint3[20743] = {X 1.9296, Y 24.2841, Z -4.6667, A 0.000, B 0.000, C 0.000 }
gfCNCPoint3[20744] = {X 1.0590, Y 23.9333, Z -4.6667, A 0.000, B 0.000, C 0.000 }
gfCNCPoint3[20745] = {X 0.2892, Y 23.3963, Z -4.6667, A 0.000, B 0.000, C 0.000 }
gfCNCPoint3[20746] = {X -0.3406, Y 22.7003, Z -4.6667, A 0.000, B 0.000, C 0.000 }
gfCNCPoint3[20747] = {X -0.7984, Y 21.8809, Z -4.6667, A 0.000, B 0.000, C 0.000 }
gfCNCPoint3[20748] = {X -3.4716, Y 15.3284, Z -4.6667, A 0.000, B 0.000, C 0.000 }
gfCNCPoint3[20749] = {X -3.6096, Y 14.8818, Z -4.6667, A 0.000, B 0.000, C 0.000 }
gfCNCPoint3[20750] = {X -3.6966, Y 14.4225, Z -4.6667, A 0.000, B 0.000, C 0.000 }
gfCNCPoint3[20751] = {X -4.2191, Y 10.4568, Z -4.6667, A 0.000, B 0.000, C 0.000 }
gfCNCPoint3[20752] = {X -7.6966, Y 10.4568, Z -4.6667, A 0.000, B 0.000, C 0.000 }
gfCNCPoint3[20753] = {X -7.6966, Y 10.4568, Z -1.6667, A 0.000, B 0.000, C 0.000 }
gfCNCPoint3[20754] = {X -7.6966, Y 10.4568, Z 11.0000, A 0.000, B 0.000, C 0.000 }
gfCNCPoint3[20755] = {X -7.9938, Y 36.0126, Z 11.0000, A 0.000, B 0.000, C 0.000 }
gfCNCPoint3[20756] = {X -7.9938, Y 36.0126, Z -1.6667, A 0.000, B 0.000, C 0.000 }
gfCNCPoint3[20757] = {X -7.9938, Y 36.0126, Z -4.6667, A 0.000, B 0.000, C 0.000 }
gfCNCPoint3[20758] = {X -4.6149, Y 35.8903, Z -4.6667, A 0.000, B 0.000, C 0.000 }
gfCNCPoint3[20759] = {X -3.6966, Y 31.9972, Z -4.6667, A 0.000, B 0.000, C 0.000 }
gfCNCPoint3[20760] = {X -3.5549, Y 31.4452, Z -4.6667, A 0.000, B 0.000, C 0.000 }
gfCNCPoint3[20761] = {X -3.3918, Y 30.8992, Z -4.6667, A 0.000, B 0.000, C 0.000 }
gfCNCPoint3[20762] = {X -3.2194, Y 30.3928, Z -4.6667, A 0.000, B 0.000, C 0.000 }
gfCNCPoint3[20763] = {X -3.0286, Y 29.8932, Z -4.6667, A 0.000, B 0.000, C 0.000 }
gfCNCPoint3[20764] = {X -2.4238, Y 28.6115, Z -4.6667, A 0.000, B 0.000, C 0.000 }
gfCNCPoint3[20765] = {X -1.6533, Y 27.4221, Z -4.6667, A 0.000, B 0.000, C 0.000 }
gfCNCPoint3[20766] = {X -0.7308, Y 26.3463, Z -4.6667, A 0.000, B 0.000, C 0.000 }
gfCNCPoint3[20767] = {X 0.3271, Y 25.4034, Z -4.6667, A 0.000, B 0.000, C 0.000 }
gfCNCPoint3[20768] = {X 1.5015, Y 24.6103, Z -4.6667, A 0.000, B 0.000, C 0.000 }
gfCNCPoint3[20769] = {X 1.8267, Y 24.4286, Z -4.6667, A 0.000, B 0.000, C 0.000 }
gfCNCPoint3[20770] = {X 2.1582, Y 24.2585, Z -4.6667, A 0.000, B 0.000, C 0.000 }
gfCNCPoint3[20771] = {X 1.2394, Y 23.9364, Z -4.6667, A 0.000, B 0.000, C 0.000 }
gfCNCPoint3[20772] = {X 0.4231, Y 23.4058, Z -4.6667, A 0.000, B 0.000, C 0.000 }
gfCNCPoint3[20773] = {X -0.2442, Y 22.6969, Z -4.6667, A 0.000, B 0.000, C 0.000 }
gfCNCPoint3[20774] = {X -0.7246, Y 21.8500, Z -4.6667, A 0.000, B 0.000, C 0.000 }
gfCNCPoint3[20775] = {X -3.3966, Y 15.3005, Z -4.6667, A 0.000, B 0.000, C 0.000 }
gfCNCPoint3[20776] = {X -3.6235, Y 14.3619, Z -4.6667, A 0.000, B 0.000, C 0.000 }
gfCNCPoint3[20777] = {X -3.6235, Y 13.3963, Z -4.6667, A 0.000, B 0.000, C 0.000 }
gfCNCPoint3[20778] = {X -3.3966, Y 12.4577, Z -4.6667, A 0.000, B 0.000, C 0.000 }
gfCNCPoint3[20779] = {X -2.9670, Y 11.6159, Z -4.6667, A 0.000, B 0.000, C 0.000 }
gfCNCPoint3[20780] = {X -2.3552, Y 10.8956, Z -4.6667, A 0.000, B 0.000, C 0.000 }
gfCNCPoint3[20781] = {X -1.5940, Y 10.3353, Z -4.6667, A 0.000, B 0.000, C 0.000 }
gfCNCPoint3[20782] = {X -0.9967, Y 9.9945, Z -4.6667, A 0.000, B 0.000, C 0.000 }
gfCNCPoint3[20783] = {X -0.1684, Y 9.6369, Z -4.6667, A 0.000, B 0.000, C 0.000 }
gfCNCPoint3[20784] = {X 0.7184, Y 9.4700, Z -4.6667, A 0.000, B 0.000, C 0.000 }
gfCNCPoint3[20785] = {X 1.6201, Y 9.5021, Z -4.6667, A 0.000, B 0.000, C 0.000 }
gfCNCPoint3[20786] = {X 2.4928, Y 9.7317, Z -4.6667, A 0.000, B 0.000, C 0.000 }
gfCNCPoint3[20787] = {X 2.5595, Y 9.7581, Z -4.6667, A 0.000, B 0.000, C 0.000 }
gfCNCPoint3[20788] = {X 2.6258, Y 9.7857, Z -4.6667, A 0.000, B 0.000, C 0.000 }
gfCNCPoint3[20789] = {X 3.4346, Y 9.3935, Z -4.6667, A 0.000, B 0.000, C 0.000 }
gfCNCPoint3[20790] = {X 4.2735, Y 9.0708, Z -4.6667, A 0.000, B 0.000, C 0.000 }
gfCNCPoint3[20791] = {X 6.1667, Y 8.4073, Z -4.6667, A 0.000, B 0.000, C 0.000 }
gfCNCPoint3[20792] = {X 8.1102, Y 7.9097, Z -4.6667, A 0.000, B 0.000, C 0.000 }
gfCNCPoint3[20793] = {X 10.0893, Y 7.5817, Z -4.6667, A 0.000, B 0.000, C 0.000 }
gfCNCPoint3[20794] = {X 12.0894, Y 7.4257, Z -4.6667, A 0.000, B 0.000, C 0.000 }
gfCNCPoint3[20795] = {X 14.0955, Y 7.4430, Z -4.6667, A 0.000, B 0.000, C 0.000 }
gfCNCPoint3[20796] = {X 16.0926, Y 7.6333, Z -4.6667, A 0.000, B 0.000, C 0.000 }
gfCNCPoint3[20797] = {X 17.8910, Y 7.9622, Z -4.6667, A 0.000, B 0.000, C 0.000 }
gfCNCPoint3[20798] = {X 19.6444, Y 8.4800, Z -4.6667, A 0.000, B 0.000, C 0.000 }
gfCNCPoint3[20799] = {X 21.3329, Y 9.1808, Z -4.6667, A 0.000, B 0.000, C 0.000 }
gfCNCPoint3[20800] = {X 22.9376, Y 10.0568, Z -4.6667, A 0.000, B 0.000, C 0.000 }
gfCNCPoint3[20801] = {X 24.4404, Y 11.0981, Z -4.6667, A 0.000, B 0.000, C 0.000 }
gfCNCPoint3[20802] = {X 25.5053, Y 12.0293, Z -4.6667, A 0.000, B 0.000, C 0.000 }
gfCNCPoint3[20803] = {X 26.4606, Y 13.0727, Z -4.6667, A 0.000, B 0.000, C 0.000 }
gfCNCPoint3[20804] = {X 27.2945, Y 14.2154, Z -4.6667, A 0.000, B 0.000, C 0.000 }
gfCNCPoint3[20805] = {X 27.9968, Y 15.4434, Z -4.6667, A 0.000, B 0.000, C 0.000 }
gfCNCPoint3[20806] = {X 28.5588, Y 16.7417, Z -4.6667, A 0.000, B 0.000, C 0.000 }
gfCNCPoint3[20807] = {X 29.0259, Y 18.3711, Z -4.6667, A 0.000, B 0.000, C 0.000 }
gfCNCPoint3[20808] = {X 29.3030, Y 20.0434, Z -4.6667, A 0.000, B 0.000, C 0.000 }
gfCNCPoint3[20809] = {X 29.3864, Y 21.7364, Z -4.6667, A 0.000, B 0.000, C 0.000 }
gfCNCPoint3[20810] = {X 29.2750, Y 23.4278, Z -4.6667, A 0.000, B 0.000, C 0.000 }
gfCNCPoint3[20811] = {X 28.9702, Y 25.0952, Z -4.6667, A 0.000, B 0.000, C 0.000 }
gfCNCPoint3[20812] = {X 28.5470, Y 26.4856, Z -4.6667, A 0.000, B 0.000, C 0.000 }
gfCNCPoint3[20813] = {X 27.9511, Y 27.8111, Z -4.6667, A 0.000, B 0.000, C 0.000 }
gfCNCPoint3[20814] = {X 27.1920, Y 29.0505, Z -4.6667, A 0.000, B 0.000, C 0.000 }
gfCNCPoint3[20815] = {X 26.2821, Y 30.1838, Z -4.6667, A 0.000, B 0.000, C 0.000 }
gfCNCPoint3[20816] = {X 25.2359, Y 31.1927, Z -4.6667, A 0.000, B 0.000, C 0.000 }
gfCNCPoint3[20817] = {X 24.9956, Y 31.3911, Z -4.6667, A 0.000, B 0.000, C 0.000 }
gfCNCPoint3[20818] = {X 24.7499, Y 31.5829, Z -4.6667, A 0.000, B 0.000, C 0.000 }
gfCNCPoint3[20819] = {X 25.6508, Y 31.8621, Z -4.6667, A 0.000, B 0.000, C 0.000 }
gfCNCPoint3[20820] = {X 26.4634, Y 32.3407, Z -4.6667, A 0.000, B 0.000, C 0.000 }
gfCNCPoint3[20821] = {X 27.1444, Y 32.9932, Z -4.6667, A 0.000, B 0.000, C 0.000 }
gfCNCPoint3[20822] = {X 27.6575, Y 33.7845, Z -4.6667, A 0.000, B 0.000, C 0.000 }
gfCNCPoint3[20823] = {X 30.6940, Y 40.0576, Z -4.6667, A 0.000, B 0.000, C 0.000 }
gfCNCPoint3[20824] = {X 30.9967, Y 40.9162, Z -4.6667, A 0.000, B 0.000, C 0.000 }
gfCNCPoint3[20825] = {X 31.1015, Y 41.8206, Z -4.6667, A 0.000, B 0.000, C 0.000 }
gfCNCPoint3[20826] = {X 31.0032, Y 42.7257, Z -4.6667, A 0.000, B 0.000, C 0.000 }
gfCNCPoint3[20827] = {X 30.7066, Y 43.5864, Z -4.6667, A 0.000, B 0.000, C 0.000 }
gfCNCPoint3[20828] = {X 30.2265, Y 44.3600, Z -4.6667, A 0.000, B 0.000, C 0.000 }
gfCNCPoint3[20829] = {X 29.5868, Y 45.0078, Z -4.6667, A 0.000, B 0.000, C 0.000 }
gfCNCPoint3[20830] = {X 29.0508, Y 45.4413, Z -4.6667, A 0.000, B 0.000, C 0.000 }
gfCNCPoint3[20831] = {X 28.3673, Y 45.8885, Z -4.6667, A 0.000, B 0.000, C 0.000 }
gfCNCPoint3[20832] = {X 27.6087, Y 46.1912, Z -4.6667, A 0.000, B 0.000, C 0.000 }
gfCNCPoint3[20833] = {X 26.8051, Y 46.3373, Z -4.6667, A 0.000, B 0.000, C 0.000 }
gfCNCPoint3[20834] = {X 25.9885, Y 46.3210, Z -4.6667, A 0.000, B 0.000, C 0.000 }
gfCNCPoint3[20835] = {X 25.1914, Y 46.1428, Z -4.6667, A 0.000, B 0.000, C 0.000 }
gfCNCPoint3[20836] = {X 23.3779, Y 47.1074, Z -4.6667, A 0.000, B 0.000, C 0.000 }
gfCNCPoint3[20837] = {X 21.5006, Y 47.9409, Z -4.6667, A 0.000, B 0.000, C 0.000 }
gfCNCPoint3[20838] = {X 19.5689, Y 48.6392, Z -4.6667, A 0.000, B 0.000, C 0.000 }
gfCNCPoint3[20839] = {X 19.4128, Y 48.6914, Z -4.6667, A 0.000, B 0.000, C 0.000 }
gfCNCPoint3[20840] = {X 17.5160, Y 49.2125, Z -4.6667, A 0.000, B 0.000, C 0.000 }
gfCNCPoint3[20841] = {X 15.5810, Y 49.5662, Z -4.6667, A 0.000, B 0.000, C 0.000 }
gfCNCPoint3[20842] = {X 13.6226, Y 49.7499, Z -4.6667, A 0.000, B 0.000, C 0.000 }
gfCNCPoint3[20843] = {X 11.6556, Y 49.7621, Z -4.6667, A 0.000, B 0.000, C 0.000 }
gfCNCPoint3[20844] = {X 9.6950, Y 49.6028, Z -4.6667, A 0.000, B 0.000, C 0.000 }
gfCNCPoint3[20845] = {X 7.7557, Y 49.2731, Z -4.6667, A 0.000, B 0.000, C 0.000 }
gfCNCPoint3[20846] = {X 5.8808, Y 48.7597, Z -4.6667, A 0.000, B 0.000, C 0.000 }
gfCNCPoint3[20847] = {X 4.0795, Y 48.0289, Z -4.6667, A 0.000, B 0.000, C 0.000 }
gfCNCPoint3[20848] = {X 2.3769, Y 47.0907, Z -4.6667, A 0.000, B 0.000, C 0.000 }
gfCNCPoint3[20849] = {X 0.7968, Y 45.9583, Z -4.6667, A 0.000, B 0.000, C 0.000 }
gfCNCPoint3[20850] = {X -0.3150, Y 44.9592, Z -4.6667, A 0.000, B 0.000, C 0.000 }
gfCNCPoint3[20851] = {X -1.3023, Y 43.8369, Z -4.6667, A 0.000, B 0.000, C 0.000 }
gfCNCPoint3[20852] = {X -2.1517, Y 42.6069, Z -4.6667, A 0.000, B 0.000, C 0.000 }
gfCNCPoint3[20853] = {X -2.8514, Y 41.2861, Z -4.6667, A 0.000, B 0.000, C 0.000 }
gfCNCPoint3[20854] = {X -3.3920, Y 39.8924, Z -4.6667, A 0.000, B 0.000, C 0.000 }
gfCNCPoint3[20855] = {X -3.5570, Y 39.3369, Z -4.6667, A 0.000, B 0.000, C 0.000 }
gfCNCPoint3[20856] = {X -3.6966, Y 38.7745, Z -4.6667, A 0.000, B 0.000, C 0.000 }
gfCNCPoint3[20857] = {X -4.5718, Y 34.8714, Z -4.6667, A 0.000, B 0.000, C 0.000 }
gfCNCPoint3[20858] = {X -7.9968, Y 34.7640, Z -4.6667, A 0.000, B 0.000, C 0.000 }
gfCNCPoint3[20859] = {X -7.9968, Y 34.7640, Z -1.6667, A 0.000, B 0.000, C 0.000 }
gfCNCPoint3[20860] = {X -7.9968, Y 34.7640, Z 11.0000, A 0.000, B 0.000, C 0.000 }
gfCNCPoint3[20861] = {X -7.9701, Y 36.4947, Z 11.0000, A 0.000, B 0.000, C 0.000 }
gfCNCPoint3[20862] = {X -7.9701, Y 36.4947, Z -1.6667, A 0.000, B 0.000, C 0.000 }
gfCNCPoint3[20863] = {X -7.9701, Y 36.4947, Z -4.6667, A 0.000, B 0.000, C 0.000 }
gfCNCPoint3[20864] = {X -4.5185, Y 36.2795, Z -4.6667, A 0.000, B 0.000, C 0.000 }
gfCNCPoint3[20865] = {X -3.6966, Y 32.3649, Z -4.6667, A 0.000, B 0.000, C 0.000 }
gfCNCPoint3[20866] = {X -3.5246, Y 31.6393, Z -4.6667, A 0.000, B 0.000, C 0.000 }
gfCNCPoint3[20867] = {X -3.3156, Y 30.9235, Z -4.6667, A 0.000, B 0.000, C 0.000 }
gfCNCPoint3[20868] = {X -3.1438, Y 30.4190, Z -4.6667, A 0.000, B 0.000, C 0.000 }
gfCNCPoint3[20869] = {X -2.9536, Y 29.9211, Z -4.6667, A 0.000, B 0.000, C 0.000 }
gfCNCPoint3[20870] = {X -2.3534, Y 28.6494, Z -4.6667, A 0.000, B 0.000, C 0.000 }
gfCNCPoint3[20871] = {X -1.5887, Y 27.4693, Z -4.6667, A 0.000, B 0.000, C 0.000 }
gfCNCPoint3[20872] = {X -0.6733, Y 26.4020, Z -4.6667, A 0.000, B 0.000, C 0.000 }
gfCNCPoint3[20873] = {X 0.3764, Y 25.4664, Z -4.6667, A 0.000, B 0.000, C 0.000 }
gfCNCPoint3[20874] = {X 1.5417, Y 24.6794, Z -4.6667, A 0.000, B 0.000, C 0.000 }
gfCNCPoint3[20875] = {X 1.9722, Y 24.4422, Z -4.6667, A 0.000, B 0.000, C 0.000 }
gfCNCPoint3[20876] = {X 2.4133, Y 24.2255, Z -4.6667, A 0.000, B 0.000, C 0.000 }
gfCNCPoint3[20877] = {X 1.6213, Y 24.0150, Z -4.6667, A 0.000, B 0.000, C 0.000 }
gfCNCPoint3[20878] = {X 0.8888, Y 23.6477, Z -4.6667, A 0.000, B 0.000, C 0.000 }
gfCNCPoint3[20879] = {X 0.2466, Y 23.1387, Z -4.6667, A 0.000, B 0.000, C 0.000 }
gfCNCPoint3[20880] = {X -0.2784, Y 22.5096, Z -4.6667, A 0.000, B 0.000, C 0.000 }
gfCNCPoint3[20881] = {X -0.6642, Y 21.7866, Z -4.6667, A 0.000, B 0.000, C 0.000 }
gfCNCPoint3[20882] = {X -3.2754, Y 15.3911, Z -4.6667, A 0.000, B 0.000, C 0.000 }
gfCNCPoint3[20883] = {X -3.2990, Y 15.3321, Z -4.6667, A 0.000, B 0.000, C 0.000 }
gfCNCPoint3[20884] = {X -3.3216, Y 15.2726, Z -4.6667, A 0.000, B 0.000, C 0.000 }
gfCNCPoint3[20885] = {X -3.5441, Y 14.3525, Z -4.6667, A 0.000, B 0.000, C 0.000 }
gfCNCPoint3[20886] = {X -3.5441, Y 13.4058, Z -4.6667, A 0.000, B 0.000, C 0.000 }
gfCNCPoint3[20887] = {X -3.3216, Y 12.4856, Z -4.6667, A 0.000, B 0.000, C 0.000 }
gfCNCPoint3[20888] = {X -2.9004, Y 11.6603, Z -4.6667, A 0.000, B 0.000, C 0.000 }
gfCNCPoint3[20889] = {X -2.3006, Y 10.9541, Z -4.6667, A 0.000, B 0.000, C 0.000 }
gfCNCPoint3[20890] = {X -1.5544, Y 10.4048, Z -4.6667, A 0.000, B 0.000, C 0.000 }
gfCNCPoint3[20891] = {X -0.9063, Y 10.0355, Z -4.6667, A 0.000, B 0.000, C 0.000 }
gfCNCPoint3[20892] = {X -0.1031, Y 9.7008, Z -4.6667, A 0.000, B 0.000, C 0.000 }
gfCNCPoint3[20893] = {X 0.7535, Y 9.5477, Z -4.6667, A 0.000, B 0.000, C 0.000 }
gfCNCPoint3[20894] = {X 1.6229, Y 9.5834, Z -4.6667, A 0.000, B 0.000, C 0.000 }
gfCNCPoint3[20895] = {X 2.4640, Y 9.8063, Z -4.6667, A 0.000, B 0.000, C 0.000 }
gfCNCPoint3[20896] = {X 2.5472, Y 9.8395, Z -4.6667, A 0.000, B 0.000, C 0.000 }
gfCNCPoint3[20897] = {X 2.6297, Y 9.8745, Z -4.6667, A 0.000, B 0.000, C 0.000 }
gfCNCPoint3[20898] = {X 3.4537, Y 9.4724, Z -4.6667, A 0.000, B 0.000, C 0.000 }
gfCNCPoint3[20899] = {X 4.3093, Y 9.1432, Z -4.6667, A 0.000, B 0.000, C 0.000 }
gfCNCPoint3[20900] = {X 6.1952, Y 8.4827, Z -4.6667, A 0.000, B 0.000, C 0.000 }
gfCNCPoint3[20901] = {X 8.1310, Y 7.9874, Z -4.6667, A 0.000, B 0.000, C 0.000 }
gfCNCPoint3[20902] = {X 10.1023, Y 7.6610, Z -4.6667, A 0.000, B 0.000, C 0.000 }
gfCNCPoint3[20903] = {X 12.0944, Y 7.5058, Z -4.6667, A 0.000, B 0.000, C 0.000 }
gfCNCPoint3[20904] = {X 14.0924, Y 7.5230, Z -4.6667, A 0.000, B 0.000, C 0.000 }
gfCNCPoint3[20905] = {X 16.0816, Y 7.7126, Z -4.6667, A 0.000, B 0.000, C 0.000 }
gfCNCPoint3[20906] = {X 16.4818, Y 7.7686, Z -4.6667, A 0.000, B 0.000, C 0.000 }
gfCNCPoint3[20907] = {X 18.1856, Y 8.1177, Z -4.6667, A 0.000, B 0.000, C 0.000 }
gfCNCPoint3[20908] = {X 19.8452, Y 8.6377, Z -4.6667, A 0.000, B 0.000, C 0.000 }
gfCNCPoint3[20909] = {X 21.4436, Y 9.3233, Z -4.6667, A 0.000, B 0.000, C 0.000 }
gfCNCPoint3[20910] = {X 22.9642, Y 10.1674, Z -4.6667, A 0.000, B 0.000, C 0.000 }
gfCNCPoint3[20911] = {X 24.3914, Y 11.1613, Z -4.6667, A 0.000, B 0.000, C 0.000 }
gfCNCPoint3[20912] = {X 25.4495, Y 12.0866, Z -4.6667, A 0.000, B 0.000, C 0.000 }
gfCNCPoint3[20913] = {X 26.3987, Y 13.1233, Z -4.6667, A 0.000, B 0.000, C 0.000 }
gfCNCPoint3[20914] = {X 27.2273, Y 14.2587, Z -4.6667, A 0.000, B 0.000, C 0.000 }
gfCNCPoint3[20915] = {X 27.9251, Y 15.4788, Z -4.6667, A 0.000, B 0.000, C 0.000 }
gfCNCPoint3[20916] = {X 28.4835, Y 16.7687, Z -4.6667, A 0.000, B 0.000, C 0.000 }
gfCNCPoint3[20917] = {X 28.9480, Y 18.3895, Z -4.6667, A 0.000, B 0.000, C 0.000 }
gfCNCPoint3[20918] = {X 29.2235, Y 20.0529, Z -4.6667, A 0.000, B 0.000, C 0.000 }
gfCNCPoint3[20919] = {X 29.3064, Y 21.7369, Z -4.6667, A 0.000, B 0.000, C 0.000 }
gfCNCPoint3[20920] = {X 29.1954, Y 23.4192, Z -4.6667, A 0.000, B 0.000, C 0.000 }
gfCNCPoint3[20921] = {X 28.8922, Y 25.0777, Z -4.6667, A 0.000, B 0.000, C 0.000 }
gfCNCPoint3[20922] = {X 28.4718, Y 26.4582, Z -4.6667, A 0.000, B 0.000, C 0.000 }
gfCNCPoint3[20923] = {X 27.8801, Y 27.7743, Z -4.6667, A 0.000, B 0.000, C 0.000 }
gfCNCPoint3[20924] = {X 27.1263, Y 29.0048, Z -4.6667, A 0.000, B 0.000, C 0.000 }
gfCNCPoint3[20925] = {X 26.2229, Y 30.1300, Z -4.6667, A 0.000, B 0.000, C 0.000 }
gfCNCPoint3[20926] = {X 25.1841, Y 31.1317, Z -4.6667, A 0.000, B 0.000, C 0.000 }
gfCNCPoint3[20927] = {X 24.8720, Y 31.3872, Z -4.6667, A 0.000, B 0.000, C 0.000 }
gfCNCPoint3[20928] = {X 24.5510, Y 31.6315, Z -4.6667, A 0.000, B 0.000, C 0.000 }
gfCNCPoint3[20929] = {X 25.3135, Y 31.8151, Z -4.6667, A 0.000, B 0.000, C 0.000 }
gfCNCPoint3[20930] = {X 26.0255, Y 32.1439, Z -4.6667, A 0.000, B 0.000, C 0.000 }
gfCNCPoint3[20931] = {X 26.6597, Y 32.6054, Z -4.6667, A 0.000, B 0.000, C 0.000 }
gfCNCPoint3[20932] = {X 27.1916, Y 33.1818, Z -4.6667, A 0.000, B 0.000, C 0.000 }
gfCNCPoint3[20933] = {X 27.6008, Y 33.8508, Z -4.6667, A 0.000, B 0.000, C 0.000 }
gfCNCPoint3[20934] = {X 30.6220, Y 40.0925, Z -4.6667, A 0.000, B 0.000, C 0.000 }
gfCNCPoint3[20935] = {X 30.9188, Y 40.9342, Z -4.6667, A 0.000, B 0.000, C 0.000 }
gfCNCPoint3[20936] = {X 31.0215, Y 41.8209, Z -4.6667, A 0.000, B 0.000, C 0.000 }
gfCNCPoint3[20937] = {X 30.9251, Y 42.7082, Z -4.6667, A 0.000, B 0.000, C 0.000 }
gfCNCPoint3[20938] = {X 30.6343, Y 43.5521, Z -4.6667, A 0.000, B 0.000, C 0.000 }
gfCNCPoint3[20939] = {X 30.1637, Y 44.3105, Z -4.6667, A 0.000, B 0.000, C 0.000 }
gfCNCPoint3[20940] = {X 29.5365, Y 44.9456, Z -4.6667, A 0.000, B 0.000, C 0.000 }
gfCNCPoint3[20941] = {X 29.0005, Y 45.3790, Z -4.6667, A 0.000, B 0.000, C 0.000 }
gfCNCPoint3[20942] = {X 28.1803, Y 45.8917, Z -4.6667, A 0.000, B 0.000, C 0.000 }
gfCNCPoint3[20943] = {X 27.2612, Y 46.1933, Z -4.6667, A 0.000, B 0.000, C 0.000 }
gfCNCPoint3[20944] = {X 26.2967, Y 46.2663, Z -4.6667, A 0.000, B 0.000, C 0.000 }
gfCNCPoint3[20945] = {X 25.3427, Y 46.1064, Z -4.6667, A 0.000, B 0.000, C 0.000 }
gfCNCPoint3[20946] = {X 25.2624, Y 46.0818, Z -4.6667, A 0.000, B 0.000, C 0.000 }
gfCNCPoint3[20947] = {X 25.1826, Y 46.0555, Z -4.6667, A 0.000, B 0.000, C 0.000 }
gfCNCPoint3[20948] = {X 23.3644, Y 47.0250, Z -4.6667, A 0.000, B 0.000, C 0.000 }
gfCNCPoint3[20949] = {X 21.4817, Y 47.8623, Z -4.6667, A 0.000, B 0.000, C 0.000 }
gfCNCPoint3[20950] = {X 19.5440, Y 48.5631, Z -4.6667, A 0.000, B 0.000, C 0.000 }
gfCNCPoint3[20951] = {X 19.3879, Y 48.6154, Z -4.6667, A 0.000, B 0.000, C 0.000 }
gfCNCPoint3[20952] = {X 17.4977, Y 49.1346, Z -4.6667, A 0.000, B 0.000, C 0.000 }
gfCNCPoint3[20953] = {X 15.5695, Y 49.4870, Z -4.6667, A 0.000, B 0.000, C 0.000 }
gfCNCPoint3[20954] = {X 13.6180, Y 49.6700, Z -4.6667, A 0.000, B 0.000, C 0.000 }
gfCNCPoint3[20955] = {X 11.6579, Y 49.6821, Z -4.6667, A 0.000, B 0.000, C 0.000 }
gfCNCPoint3[20956] = {X 9.7042, Y 49.5233, Z -4.6667, A 0.000, B 0.000, C 0.000 }
gfCNCPoint3[20957] = {X 7.7718, Y 49.1947, Z -4.6667, A 0.000, B 0.000, C 0.000 }
gfCNCPoint3[20958] = {X 5.9057, Y 48.6837, Z -4.6667, A 0.000, B 0.000, C 0.000 }
gfCNCPoint3[20959] = {X 4.1128, Y 47.9562, Z -4.6667, A 0.000, B 0.000, C 0.000 }
gfCNCPoint3[20960] = {X 2.4183, Y 47.0223, Z -4.6667, A 0.000, B 0.000, C 0.000 }
gfCNCPoint3[20961] = {X 0.8458, Y 45.8951, Z -4.6667, A 0.000, B 0.000, C 0.000 }
gfCNCPoint3[20962] = {X -0.2588, Y 44.9023, Z -4.6667, A 0.000, B 0.000, C 0.000 }
gfCNCPoint3[20963] = {X -1.2397, Y 43.7871, Z -4.6667, A 0.000, B 0.000, C 0.000 }
gfCNCPoint3[20964] = {X -2.0835, Y 42.5650, Z -4.6667, A 0.000, B 0.000, C 0.000 }
gfCNCPoint3[20965] = {X -2.7788, Y 41.2526, Z -4.6667, A 0.000, B 0.000, C 0.000 }
gfCNCPoint3[20966] = {X -3.3158, Y 39.8679, Z -4.6667, A 0.000, B 0.000, C 0.000 }
gfCNCPoint3[20967] = {X -3.5287, Y 39.1310, Z -4.6667, A 0.000, B 0.000, C 0.000 }
gfCNCPoint3[20968] = {X -3.6966, Y 38.3825, Z -4.6667, A 0.000, B 0.000, C 0.000 }
gfCNCPoint3[20969] = {X -4.4537, Y 34.4548, Z -4.6667, A 0.000, B 0.000, C 0.000 }
gfCNCPoint3[20970] = {X -7.9733, Y 34.2455, Z -4.6667, A 0.000, B 0.000, C 0.000 }
gfCNCPoint3[20971] = {X -7.9733, Y 34.2455, Z -1.6667, A 0.000, B 0.000, C 0.000 }
gfCNCPoint3[20972] = {X -7.9733, Y 34.2455, Z 11.0000, A 0.000, B 0.000, C 0.000 }
gfCNCPoint3[20973] = {X 39.8249, Y 26.3830, Z 11.0000, A 0.000, B 0.000, C 0.000 }
gfCNCPoint3[20974] = {X 39.8249, Y 26.3830, Z -1.6667, A 0.000, B 0.000, C 0.000 }
gfCNCPoint3[20975] = {X 39.8249, Y 26.3830, Z -4.6667, A 0.000, B 0.000, C 0.000 }
gfCNCPoint3[20976] = {X 43.6483, Y 27.8071, Z -4.6667, A 0.000, B 0.000, C 0.000 }
gfCNCPoint3[20977] = {X 48.2901, Y 15.3446, Z -4.6667, A 0.000, B 0.000, C 0.000 }
gfCNCPoint3[20978] = {X 47.9078, Y 14.6186, Z -4.6667, A 0.000, B 0.000, C 0.000 }
gfCNCPoint3[20979] = {X 47.6697, Y 13.8333, Z -4.6667, A 0.000, B 0.000, C 0.000 }
gfCNCPoint3[20980] = {X 47.5844, Y 13.0172, Z -4.6667, A 0.000, B 0.000, C 0.000 }
gfCNCPoint3[20981] = {X 47.5842, Y 12.1868, Z -4.6667, A 0.000, B 0.000, C 0.000 }
gfCNCPoint3[20982] = {X 47.6925, Y 11.2255, Z -4.6667, A 0.000, B 0.000, C 0.000 }
gfCNCPoint3[20983] = {X 48.0120, Y 10.3125, Z -4.6667, A 0.000, B 0.000, C 0.000 }
gfCNCPoint3[20984] = {X 48.5267, Y 9.4933, Z -4.6667, A 0.000, B 0.000, C 0.000 }
gfCNCPoint3[20985] = {X 49.2107, Y 8.8093, Z -4.6667, A 0.000, B 0.000, C 0.000 }
gfCNCPoint3[20986] = {X 50.0298, Y 8.2946, Z -4.6667, A 0.000, B 0.000, C 0.000 }
gfCNCPoint3[20987] = {X 50.9429, Y 7.9751, Z -4.6667, A 0.000, B 0.000, C 0.000 }
gfCNCPoint3[20988] = {X 51.9042, Y 7.8668, Z -4.6667, A 0.000, B 0.000, C 0.000 }
gfCNCPoint3[20989] = {X 59.6221, Y 7.8668, Z -4.6667, A 0.000, B 0.000, C 0.000 }
gfCNCPoint3[20990] = {X 60.5834, Y 7.9751, Z -4.6667, A 0.000, B 0.000, C 0.000 }
gfCNCPoint3[20991] = {X 61.4965, Y 8.2946, Z -4.6667, A 0.000, B 0.000, C 0.000 }
gfCNCPoint3[20992] = {X 62.3156, Y 8.8093, Z -4.6667, A 0.000, B 0.000, C 0.000 }
gfCNCPoint3[20993] = {X 62.9996, Y 9.4933, Z -4.6667, A 0.000, B 0.000, C 0.000 }
gfCNCPoint3[20994] = {X 63.5143, Y 10.3124, Z -4.6667, A 0.000, B 0.000, C 0.000 }
gfCNCPoint3[20995] = {X 63.8338, Y 11.2255, Z -4.6667, A 0.000, B 0.000, C 0.000 }
gfCNCPoint3[20996] = {X 63.9421, Y 12.1868, Z -4.6667, A 0.000, B 0.000, C 0.000 }
gfCNCPoint3[20997] = {X 63.9421, Y 12.9782, Z -4.6667, A 0.000, B 0.000, C 0.000 }
gfCNCPoint3[20998] = {X 63.8583, Y 13.8247, Z -4.6667, A 0.000, B 0.000, C 0.000 }
gfCNCPoint3[20999] = {X 63.6103, Y 14.6384, Z -4.6667, A 0.000, B 0.000, C 0.000 }
gfCNCPoint3[21000] = {X 63.2077, Y 15.3877, Z -4.6667, A 0.000, B 0.000, C 0.000 }
gfCNCPoint3[21001] = {X 63.4258, Y 15.9633, Z -4.6667, A 0.000, B 0.000, C 0.000 }
gfCNCPoint3[21002] = {X 66.2401, Y 23.4311, Z -4.6667, A 0.000, B 0.000, C 0.000 }
gfCNCPoint3[21003] = {X 72.2097, Y 39.5004, Z -4.6667, A 0.000, B 0.000, C 0.000 }
gfCNCPoint3[21004] = {X 72.5150, Y 40.2683, Z -4.6667, A 0.000, B 0.000, C 0.000 }
gfCNCPoint3[21005] = {X 73.3594, Y 40.7701, Z -4.6667, A 0.000, B 0.000, C 0.000 }
gfCNCPoint3[21006] = {X 74.0686, Y 41.4497, Z -4.6667, A 0.000, B 0.000, C 0.000 }
gfCNCPoint3[21007] = {X 74.6059, Y 42.2719, Z -4.6667, A 0.000, B 0.000, C 0.000 }
gfCNCPoint3[21008] = {X 74.9437, Y 43.1943, Z -4.6667, A 0.000, B 0.000, C 0.000 }
gfCNCPoint3[21009] = {X 75.0643, Y 44.1692, Z -4.6667, A 0.000, B 0.000, C 0.000 }
gfCNCPoint3[21010] = {X 75.0645, Y 45.0000, Z -4.6667, A 0.000, B 0.000, C 0.000 }
gfCNCPoint3[21011] = {X 74.9561, Y 45.9613, Z -4.6667, A 0.000, B 0.000, C 0.000 }
gfCNCPoint3[21012] = {X 74.6366, Y 46.8744, Z -4.6667, A 0.000, B 0.000, C 0.000 }
gfCNCPoint3[21013] = {X 74.1220, Y 47.6935, Z -4.6667, A 0.000, B 0.000, C 0.000 }
gfCNCPoint3[21014] = {X 73.4379, Y 48.3775, Z -4.6667, A 0.000, B 0.000, C 0.000 }
gfCNCPoint3[21015] = {X 72.6188, Y 48.8922, Z -4.6667, A 0.000, B 0.000, C 0.000 }
gfCNCPoint3[21016] = {X 71.7057, Y 49.2117, Z -4.6667, A 0.000, B 0.000, C 0.000 }
gfCNCPoint3[21017] = {X 70.7445, Y 49.3200, Z -4.6667, A 0.000, B 0.000, C 0.000 }
gfCNCPoint3[21018] = {X 64.1851, Y 49.3200, Z -4.6667, A 0.000, B 0.000, C 0.000 }
gfCNCPoint3[21019] = {X 63.2238, Y 49.2117, Z -4.6667, A 0.000, B 0.000, C 0.000 }
gfCNCPoint3[21020] = {X 62.3108, Y 48.8922, Z -4.6667, A 0.000, B 0.000, C 0.000 }
gfCNCPoint3[21021] = {X 61.4917, Y 48.3775, Z -4.6667, A 0.000, B 0.000, C 0.000 }
gfCNCPoint3[21022] = {X 60.8076, Y 47.6935, Z -4.6667, A 0.000, B 0.000, C 0.000 }
gfCNCPoint3[21023] = {X 60.2929, Y 46.8744, Z -4.6667, A 0.000, B 0.000, C 0.000 }
gfCNCPoint3[21024] = {X 59.9734, Y 45.9613, Z -4.6667, A 0.000, B 0.000, C 0.000 }
gfCNCPoint3[21025] = {X 59.8651, Y 45.0000, Z -4.6667, A 0.000, B 0.000, C 0.000 }
gfCNCPoint3[21026] = {X 59.8651, Y 44.2085, Z -4.6667, A 0.000, B 0.000, C 0.000 }
gfCNCPoint3[21027] = {X 59.9518, Y 43.3501, Z -4.6667, A 0.000, B 0.000, C 0.000 }
gfCNCPoint3[21028] = {X 60.2074, Y 42.5261, Z -4.6667, A 0.000, B 0.000, C 0.000 }
gfCNCPoint3[21029] = {X 60.6216, Y 41.7693, Z -4.6667, A 0.000, B 0.000, C 0.000 }
gfCNCPoint3[21030] = {X 60.0069, Y 40.0892, Z -4.6667, A 0.000, B 0.000, C 0.000 }
gfCNCPoint3[21031] = {X 52.0773, Y 40.0892, Z -4.6667, A 0.000, B 0.000, C 0.000 }
gfCNCPoint3[21032] = {X 51.3345, Y 42.0848, Z -4.6667, A 0.000, B 0.000, C 0.000 }
gfCNCPoint3[21033] = {X 51.3376, Y 42.0899, Z -4.6667, A 0.000, B 0.000, C 0.000 }
gfCNCPoint3[21034] = {X 51.6390, Y 42.7494, Z -4.6667, A 0.000, B 0.000, C 0.000 }
gfCNCPoint3[21035] = {X 51.8258, Y 43.4500, Z -4.6667, A 0.000, B 0.000, C 0.000 }
gfCNCPoint3[21036] = {X 51.8928, Y 44.1720, Z -4.6667, A 0.000, B 0.000, C 0.000 }
gfCNCPoint3[21037] = {X 51.8929, Y 45.0000, Z -4.6667, A 0.000, B 0.000, C 0.000 }
gfCNCPoint3[21038] = {X 51.7846, Y 45.9613, Z -4.6667, A 0.000, B 0.000, C 0.000 }
gfCNCPoint3[21039] = {X 51.4651, Y 46.8744, Z -4.6667, A 0.000, B 0.000, C 0.000 }
gfCNCPoint3[21040] = {X 50.9504, Y 47.6935, Z -4.6667, A 0.000, B 0.000, C 0.000 }
gfCNCPoint3[21041] = {X 50.2664, Y 48.3775, Z -4.6667, A 0.000, B 0.000, C 0.000 }
gfCNCPoint3[21042] = {X 49.4473, Y 48.8922, Z -4.6667, A 0.000, B 0.000, C 0.000 }
gfCNCPoint3[21043] = {X 48.5342, Y 49.2117, Z -4.6667, A 0.000, B 0.000, C 0.000 }
gfCNCPoint3[21044] = {X 47.5729, Y 49.3200, Z -4.6667, A 0.000, B 0.000, C 0.000 }
gfCNCPoint3[21045] = {X 40.6393, Y 49.3200, Z -4.6667, A 0.000, B 0.000, C 0.000 }
gfCNCPoint3[21046] = {X 39.6780, Y 49.2117, Z -4.6667, A 0.000, B 0.000, C 0.000 }
gfCNCPoint3[21047] = {X 38.7649, Y 48.8922, Z -4.6667, A 0.000, B 0.000, C 0.000 }
gfCNCPoint3[21048] = {X 37.9458, Y 48.3775, Z -4.6667, A 0.000, B 0.000, C 0.000 }
gfCNCPoint3[21049] = {X 37.2618, Y 47.6935, Z -4.6667, A 0.000, B 0.000, C 0.000 }
gfCNCPoint3[21050] = {X 36.7471, Y 46.8744, Z -4.6667, A 0.000, B 0.000, C 0.000 }
gfCNCPoint3[21051] = {X 36.4276, Y 45.9613, Z -4.6667, A 0.000, B 0.000, C 0.000 }
gfCNCPoint3[21052] = {X 36.3193, Y 45.0000, Z -4.6667, A 0.000, B 0.000, C 0.000 }
gfCNCPoint3[21053] = {X 36.3193, Y 44.2086, Z -4.6667, A 0.000, B 0.000, C 0.000 }
gfCNCPoint3[21054] = {X 36.4360, Y 43.2115, Z -4.6667, A 0.000, B 0.000, C 0.000 }
gfCNCPoint3[21055] = {X 36.7797, Y 42.2682, Z -4.6667, A 0.000, B 0.000, C 0.000 }
gfCNCPoint3[21056] = {X 37.3319, Y 41.4297, Z -4.6667, A 0.000, B 0.000, C 0.000 }
gfCNCPoint3[21057] = {X 38.0627, Y 40.7413, Z -4.6667, A 0.000, B 0.000, C 0.000 }
gfCNCPoint3[21058] = {X 38.9326, Y 40.2402, Z -4.6667, A 0.000, B 0.000, C 0.000 }
gfCNCPoint3[21059] = {X 39.5235, Y 38.8449, Z -4.6667, A 0.000, B 0.000, C 0.000 }
gfCNCPoint3[21060] = {X 40.0643, Y 37.4294, Z -4.6667, A 0.000, B 0.000, C 0.000 }
gfCNCPoint3[21061] = {X 43.6483, Y 27.8071, Z -4.6667, A 0.000, B 0.000, C 0.000 }
gfCNCPoint3[21062] = {X 39.8999, Y 26.4109, Z -4.6667, A 0.000, B 0.000, C 0.000 }
gfCNCPoint3[21063] = {X 43.7233, Y 27.8350, Z -4.6667, A 0.000, B 0.000, C 0.000 }
gfCNCPoint3[21064] = {X 48.3793, Y 15.3344, Z -4.6667, A 0.000, B 0.000, C 0.000 }
gfCNCPoint3[21065] = {X 47.9921, Y 14.6130, Z -4.6667, A 0.000, B 0.000, C 0.000 }
gfCNCPoint3[21066] = {X 47.7508, Y 13.8306, Z -4.6667, A 0.000, B 0.000, C 0.000 }
gfCNCPoint3[21067] = {X 47.6644, Y 13.0164, Z -4.6667, A 0.000, B 0.000, C 0.000 }
gfCNCPoint3[21068] = {X 47.6642, Y 12.1868, Z -4.6667, A 0.000, B 0.000, C 0.000 }
gfCNCPoint3[21069] = {X 47.7705, Y 11.2433, Z -4.6667, A 0.000, B 0.000, C 0.000 }
gfCNCPoint3[21070] = {X 48.0841, Y 10.3472, Z -4.6667, A 0.000, B 0.000, C 0.000 }
gfCNCPoint3[21071] = {X 48.5893, Y 9.5432, Z -4.6667, A 0.000, B 0.000, C 0.000 }
gfCNCPoint3[21072] = {X 49.2606, Y 8.8719, Z -4.6667, A 0.000, B 0.000, C 0.000 }
gfCNCPoint3[21073] = {X 50.0646, Y 8.3667, Z -4.6667, A 0.000, B 0.000, C 0.000 }
gfCNCPoint3[21074] = {X 50.9607, Y 8.0531, Z -4.6667, A 0.000, B 0.000, C 0.000 }
gfCNCPoint3[21075] = {X 51.9042, Y 7.9468, Z -4.6667, A 0.000, B 0.000, C 0.000 }
gfCNCPoint3[21076] = {X 59.6221, Y 7.9468, Z -4.6667, A 0.000, B 0.000, C 0.000 }
gfCNCPoint3[21077] = {X 60.5656, Y 8.0531, Z -4.6667, A 0.000, B 0.000, C 0.000 }
gfCNCPoint3[21078] = {X 61.4618, Y 8.3667, Z -4.6667, A 0.000, B 0.000, C 0.000 }
gfCNCPoint3[21079] = {X 62.2657, Y 8.8718, Z -4.6667, A 0.000, B 0.000, C 0.000 }
gfCNCPoint3[21080] = {X 62.9371, Y 9.5432, Z -4.6667, A 0.000, B 0.000, C 0.000 }
gfCNCPoint3[21081] = {X 63.4422, Y 10.3471, Z -4.6667, A 0.000, B 0.000, C 0.000 }
gfCNCPoint3[21082] = {X 63.7558, Y 11.2433, Z -4.6667, A 0.000, B 0.000, C 0.000 }
gfCNCPoint3[21083] = {X 63.8621, Y 12.1868, Z -4.6667, A 0.000, B 0.000, C 0.000 }
gfCNCPoint3[21084] = {X 63.8621, Y 12.9781, Z -4.6667, A 0.000, B 0.000, C 0.000 }
gfCNCPoint3[21085] = {X 63.7772, Y 13.8225, Z -4.6667, A 0.000, B 0.000, C 0.000 }
gfCNCPoint3[21086] = {X 63.5258, Y 14.6329, Z -4.6667, A 0.000, B 0.000, C 0.000 }
gfCNCPoint3[21087] = {X 63.1181, Y 15.3771, Z -4.6667, A 0.000, B 0.000, C 0.000 }
gfCNCPoint3[21088] = {X 63.3510, Y 15.9916, Z -4.6667, A 0.000, B 0.000, C 0.000 }
gfCNCPoint3[21089] = {X 66.1652, Y 23.4592, Z -4.6667, A 0.000, B 0.000, C 0.000 }
gfCNCPoint3[21090] = {X 72.1350, Y 39.5291, Z -4.6667, A 0.000, B 0.000, C 0.000 }
gfCNCPoint3[21091] = {X 72.4527, Y 40.3281, Z -4.6667, A 0.000, B 0.000, C 0.000 }
gfCNCPoint3[21092] = {X 73.2903, Y 40.8182, Z -4.6667, A 0.000, B 0.000, C 0.000 }
gfCNCPoint3[21093] = {X 73.9946, Y 41.4859, Z -4.6667, A 0.000, B 0.000, C 0.000 }
gfCNCPoint3[21094] = {X 74.5286, Y 42.2963, Z -4.6667, A 0.000, B 0.000, C 0.000 }
gfCNCPoint3[21095] = {X 74.8644, Y 43.2068, Z -4.6667, A 0.000, B 0.000, C 0.000 }
gfCNCPoint3[21096] = {X 74.9843, Y 44.1699, Z -4.6667, A 0.000, B 0.000, C 0.000 }
gfCNCPoint3[21097] = {X 74.9845, Y 45.0000, Z -4.6667, A 0.000, B 0.000, C 0.000 }
gfCNCPoint3[21098] = {X 74.8782, Y 45.9435, Z -4.6667, A 0.000, B 0.000, C 0.000 }
gfCNCPoint3[21099] = {X 74.5646, Y 46.8397, Z -4.6667, A 0.000, B 0.000, C 0.000 }
gfCNCPoint3[21100] = {X 74.0594, Y 47.6436, Z -4.6667, A 0.000, B 0.000, C 0.000 }
gfCNCPoint3[21101] = {X 73.3881, Y 48.3150, Z -4.6667, A 0.000, B 0.000, C 0.000 }
gfCNCPoint3[21102] = {X 72.5841, Y 48.8201, Z -4.6667, A 0.000, B 0.000, C 0.000 }
gfCNCPoint3[21103] = {X 71.6879, Y 49.1337, Z -4.6667, A 0.000, B 0.000, C 0.000 }
gfCNCPoint3[21104] = {X 70.7445, Y 49.2400, Z -4.6667, A 0.000, B 0.000, C 0.000 }
gfCNCPoint3[21105] = {X 64.1851, Y 49.2400, Z -4.6667, A 0.000, B 0.000, C 0.000 }
gfCNCPoint3[21106] = {X 63.2416, Y 49.1337, Z -4.6667, A 0.000, B 0.000, C 0.000 }
gfCNCPoint3[21107] = {X 62.3455, Y 48.8201, Z -4.6667, A 0.000, B 0.000, C 0.000 }
gfCNCPoint3[21108] = {X 61.5415, Y 48.3150, Z -4.6667, A 0.000, B 0.000, C 0.000 }
gfCNCPoint3[21109] = {X 60.8702, Y 47.6436, Z -4.6667, A 0.000, B 0.000, C 0.000 }
gfCNCPoint3[21110] = {X 60.3650, Y 46.8397, Z -4.6667, A 0.000, B 0.000, C 0.000 }
gfCNCPoint3[21111] = {X 60.0514, Y 45.9435, Z -4.6667, A 0.000, B 0.000, C 0.000 }
gfCNCPoint3[21112] = {X 59.9451, Y 45.0000, Z -4.6667, A 0.000, B 0.000, C 0.000 }
gfCNCPoint3[21113] = {X 59.9451, Y 44.2085, Z -4.6667, A 0.000, B 0.000, C 0.000 }
gfCNCPoint3[21114] = {X 60.0330, Y 43.3526, Z -4.6667, A 0.000, B 0.000, C 0.000 }
gfCNCPoint3[21115] = {X 60.2918, Y 42.5321, Z -4.6667, A 0.000, B 0.000, C 0.000 }
gfCNCPoint3[21116] = {X 60.7110, Y 41.7807, Z -4.6667, A 0.000, B 0.000, C 0.000 }
gfCNCPoint3[21117] = {X 60.0628, Y 40.0092, Z -4.6667, A 0.000, B 0.000, C 0.000 }
gfCNCPoint3[21118] = {X 52.0217, Y 40.0092, Z -4.6667, A 0.000, B 0.000, C 0.000 }
gfCNCPoint3[21119] = {X 51.2461, Y 42.0930, Z -4.6667, A 0.000, B 0.000, C 0.000 }
gfCNCPoint3[21120] = {X 51.2684, Y 42.1301, Z -4.6667, A 0.000, B 0.000, C 0.000 }
gfCNCPoint3[21121] = {X 51.5639, Y 42.7771, Z -4.6667, A 0.000, B 0.000, C 0.000 }
gfCNCPoint3[21122] = {X 51.7471, Y 43.4644, Z -4.6667, A 0.000, B 0.000, C 0.000 }
gfCNCPoint3[21123] = {X 51.8128, Y 44.1726, Z -4.6667, A 0.000, B 0.000, C 0.000 }
gfCNCPoint3[21124] = {X 51.8129, Y 45.0000, Z -4.6667, A 0.000, B 0.000, C 0.000 }
gfCNCPoint3[21125] = {X 51.7066, Y 45.9435, Z -4.6667, A 0.000, B 0.000, C 0.000 }
gfCNCPoint3[21126] = {X 51.3930, Y 46.8397, Z -4.6667, A 0.000, B 0.000, C 0.000 }
gfCNCPoint3[21127] = {X 50.8879, Y 47.6436, Z -4.6667, A 0.000, B 0.000, C 0.000 }
gfCNCPoint3[21128] = {X 50.2165, Y 48.3150, Z -4.6667, A 0.000, B 0.000, C 0.000 }
gfCNCPoint3[21129] = {X 49.4126, Y 48.8201, Z -4.6667, A 0.000, B 0.000, C 0.000 }
gfCNCPoint3[21130] = {X 48.5164, Y 49.1337, Z -4.6667, A 0.000, B 0.000, C 0.000 }
gfCNCPoint3[21131] = {X 47.5729, Y 49.2400, Z -4.6667, A 0.000, B 0.000, C 0.000 }
gfCNCPoint3[21132] = {X 40.6393, Y 49.2400, Z -4.6667, A 0.000, B 0.000, C 0.000 }
gfCNCPoint3[21133] = {X 39.6958, Y 49.1337, Z -4.6667, A 0.000, B 0.000, C 0.000 }
gfCNCPoint3[21134] = {X 38.7996, Y 48.8201, Z -4.6667, A 0.000, B 0.000, C 0.000 }
gfCNCPoint3[21135] = {X 37.9957, Y 48.3150, Z -4.6667, A 0.000, B 0.000, C 0.000 }
gfCNCPoint3[21136] = {X 37.3243, Y 47.6436, Z -4.6667, A 0.000, B 0.000, C 0.000 }
gfCNCPoint3[21137] = {X 36.8192, Y 46.8397, Z -4.6667, A 0.000, B 0.000, C 0.000 }
gfCNCPoint3[21138] = {X 36.5056, Y 45.9435, Z -4.6667, A 0.000, B 0.000, C 0.000 }
gfCNCPoint3[21139] = {X 36.3993, Y 45.0000, Z -4.6667, A 0.000, B 0.000, C 0.000 }
gfCNCPoint3[21140] = {X 36.3993, Y 44.2086, Z -4.6667, A 0.000, B 0.000, C 0.000 }
gfCNCPoint3[21141] = {X 36.5153, Y 43.2239, Z -4.6667, A 0.000, B 0.000, C 0.000 }
gfCNCPoint3[21142] = {X 36.8568, Y 42.2930, Z -4.6667, A 0.000, B 0.000, C 0.000 }
gfCNCPoint3[21143] = {X 37.4052, Y 41.4669, Z -4.6667, A 0.000, B 0.000, C 0.000 }
gfCNCPoint3[21144] = {X 38.1304, Y 40.7907, Z -4.6667, A 0.000, B 0.000, C 0.000 }
gfCNCPoint3[21145] = {X 38.9929, Y 40.3015, Z -4.6667, A 0.000, B 0.000, C 0.000 }
gfCNCPoint3[21146] = {X 39.5918, Y 38.8894, Z -4.6667, A 0.000, B 0.000, C 0.000 }
gfCNCPoint3[21147] = {X 40.1396, Y 37.4566, Z -4.6667, A 0.000, B 0.000, C 0.000 }
gfCNCPoint3[21148] = {X 43.7233, Y 27.8350, Z -4.6667, A 0.000, B 0.000, C 0.000 }
gfCNCPoint3[21149] = {X 39.9749, Y 26.4388, Z -4.6667, A 0.000, B 0.000, C 0.000 }
gfCNCPoint3[21150] = {X 43.7983, Y 27.8629, Z -4.6667, A 0.000, B 0.000, C 0.000 }
gfCNCPoint3[21151] = {X 48.4687, Y 15.3238, Z -4.6667, A 0.000, B 0.000, C 0.000 }
gfCNCPoint3[21152] = {X 48.0765, Y 14.6072, Z -4.6667, A 0.000, B 0.000, C 0.000 }
gfCNCPoint3[21153] = {X 47.8320, Y 13.8278, Z -4.6667, A 0.000, B 0.000, C 0.000 }
gfCNCPoint3[21154] = {X 47.7444, Y 13.0157, Z -4.6667, A 0.000, B 0.000, C 0.000 }
gfCNCPoint3[21155] = {X 47.7442, Y 12.1868, Z -4.6667, A 0.000, B 0.000, C 0.000 }
gfCNCPoint3[21156] = {X 47.8485, Y 11.2611, Z -4.6667, A 0.000, B 0.000, C 0.000 }
gfCNCPoint3[21157] = {X 48.1562, Y 10.3819, Z -4.6667, A 0.000, B 0.000, C 0.000 }
gfCNCPoint3[21158] = {X 48.6518, Y 9.5931, Z -4.6667, A 0.000, B 0.000, C 0.000 }
gfCNCPoint3[21159] = {X 49.3105, Y 8.9344, Z -4.6667, A 0.000, B 0.000, C 0.000 }
gfCNCPoint3[21160] = {X 50.0993, Y 8.4388, Z -4.6667, A 0.000, B 0.000, C 0.000 }
gfCNCPoint3[21161] = {X 50.9785, Y 8.1311, Z -4.6667, A 0.000, B 0.000, C 0.000 }
gfCNCPoint3[21162] = {X 51.9042, Y 8.0268, Z -4.6667, A 0.000, B 0.000, C 0.000 }
gfCNCPoint3[21163] = {X 59.6221, Y 8.0268, Z -4.6667, A 0.000, B 0.000, C 0.000 }
gfCNCPoint3[21164] = {X 60.5478, Y 8.1311, Z -4.6667, A 0.000, B 0.000, C 0.000 }
gfCNCPoint3[21165] = {X 61.4271, Y 8.4388, Z -4.6667, A 0.000, B 0.000, C 0.000 }
gfCNCPoint3[21166] = {X 62.2158, Y 8.9344, Z -4.6667, A 0.000, B 0.000, C 0.000 }
gfCNCPoint3[21167] = {X 62.8745, Y 9.5931, Z -4.6667, A 0.000, B 0.000, C 0.000 }
gfCNCPoint3[21168] = {X 63.3702, Y 10.3819, Z -4.6667, A 0.000, B 0.000, C 0.000 }
gfCNCPoint3[21169] = {X 63.6778, Y 11.2611, Z -4.6667, A 0.000, B 0.000, C 0.000 }
gfCNCPoint3[21170] = {X 63.7821, Y 12.1868, Z -4.6667, A 0.000, B 0.000, C 0.000 }
gfCNCPoint3[21171] = {X 63.7821, Y 12.9781, Z -4.6667, A 0.000, B 0.000, C 0.000 }
gfCNCPoint3[21172] = {X 63.6960, Y 13.8201, Z -4.6667, A 0.000, B 0.000, C 0.000 }
gfCNCPoint3[21173] = {X 63.4412, Y 14.6273, Z -4.6667, A 0.000, B 0.000, C 0.000 }
gfCNCPoint3[21174] = {X 63.0284, Y 15.3661, Z -4.6667, A 0.000, B 0.000, C 0.000 }
gfCNCPoint3[21175] = {X 63.2761, Y 16.0199, Z -4.6667, A 0.000, B 0.000, C 0.000 }
gfCNCPoint3[21176] = {X 66.0903, Y 23.4872, Z -4.6667, A 0.000, B 0.000, C 0.000 }
gfCNCPoint3[21177] = {X 72.0603, Y 39.5578, Z -4.6667, A 0.000, B 0.000, C 0.000 }
gfCNCPoint3[21178] = {X 72.3905, Y 40.3883, Z -4.6667, A 0.000, B 0.000, C 0.000 }
gfCNCPoint3[21179] = {X 73.2214, Y 40.8666, Z -4.6667, A 0.000, B 0.000, C 0.000 }
gfCNCPoint3[21180] = {X 73.9207, Y 41.5223, Z -4.6667, A 0.000, B 0.000, C 0.000 }
gfCNCPoint3[21181] = {X 74.4513, Y 42.3207, Z -4.6667, A 0.000, B 0.000, C 0.000 }
gfCNCPoint3[21182] = {X 74.7851, Y 43.2194, Z -4.6667, A 0.000, B 0.000, C 0.000 }
gfCNCPoint3[21183] = {X 74.9043, Y 44.1706, Z -4.6667, A 0.000, B 0.000, C 0.000 }
gfCNCPoint3[21184] = {X 74.9045, Y 45.0000, Z -4.6667, A 0.000, B 0.000, C 0.000 }
gfCNCPoint3[21185] = {X 74.8002, Y 45.9257, Z -4.6667, A 0.000, B 0.000, C 0.000 }
gfCNCPoint3[21186] = {X 74.4925, Y 46.8050, Z -4.6667, A 0.000, B 0.000, C 0.000 }
gfCNCPoint3[21187] = {X 73.9969, Y 47.5937, Z -4.6667, A 0.000, B 0.000, C 0.000 }
gfCNCPoint3[21188] = {X 73.3382, Y 48.2524, Z -4.6667, A 0.000, B 0.000, C 0.000 }
gfCNCPoint3[21189] = {X 72.5494, Y 48.7480, Z -4.6667, A 0.000, B 0.000, C 0.000 }
gfCNCPoint3[21190] = {X 71.6701, Y 49.0557, Z -4.6667, A 0.000, B 0.000, C 0.000 }
gfCNCPoint3[21191] = {X 70.7445, Y 49.1600, Z -4.6667, A 0.000, B 0.000, C 0.000 }
gfCNCPoint3[21192] = {X 64.1851, Y 49.1600, Z -4.6667, A 0.000, B 0.000, C 0.000 }
gfCNCPoint3[21193] = {X 63.2594, Y 49.0557, Z -4.6667, A 0.000, B 0.000, C 0.000 }
gfCNCPoint3[21194] = {X 62.3802, Y 48.7480, Z -4.6667, A 0.000, B 0.000, C 0.000 }
gfCNCPoint3[21195] = {X 61.5914, Y 48.2524, Z -4.6667, A 0.000, B 0.000, C 0.000 }
gfCNCPoint3[21196] = {X 60.9327, Y 47.5937, Z -4.6667, A 0.000, B 0.000, C 0.000 }
gfCNCPoint3[21197] = {X 60.4371, Y 46.8050, Z -4.6667, A 0.000, B 0.000, C 0.000 }
gfCNCPoint3[21198] = {X 60.1294, Y 45.9257, Z -4.6667, A 0.000, B 0.000, C 0.000 }
gfCNCPoint3[21199] = {X 60.0251, Y 45.0000, Z -4.6667, A 0.000, B 0.000, C 0.000 }
gfCNCPoint3[21200] = {X 60.0251, Y 44.2086, Z -4.6667, A 0.000, B 0.000, C 0.000 }
gfCNCPoint3[21201] = {X 60.1142, Y 43.3553, Z -4.6667, A 0.000, B 0.000, C 0.000 }
gfCNCPoint3[21202] = {X 60.3763, Y 42.5384, Z -4.6667, A 0.000, B 0.000, C 0.000 }
gfCNCPoint3[21203] = {X 60.8005, Y 41.7927, Z -4.6667, A 0.000, B 0.000, C 0.000 }
gfCNCPoint3[21204] = {X 60.1188, Y 39.9292, Z -4.6667, A 0.000, B 0.000, C 0.000 }
gfCNCPoint3[21205] = {X 51.9662, Y 39.9292, Z -4.6667, A 0.000, B 0.000, C 0.000 }
gfCNCPoint3[21206] = {X 51.1577, Y 42.1011, Z -4.6667, A 0.000, B 0.000, C 0.000 }
gfCNCPoint3[21207] = {X 51.1992, Y 42.1703, Z -4.6667, A 0.000, B 0.000, C 0.000 }
gfCNCPoint3[21208] = {X 51.4889, Y 42.8048, Z -4.6667, A 0.000, B 0.000, C 0.000 }
gfCNCPoint3[21209] = {X 51.6684, Y 43.4788, Z -4.6667, A 0.000, B 0.000, C 0.000 }
gfCNCPoint3[21210] = {X 51.7328, Y 44.1733, Z -4.6667, A 0.000, B 0.000, C 0.000 }
gfCNCPoint3[21211] = {X 51.7329, Y 45.0000, Z -4.6667, A 0.000, B 0.000, C 0.000 }
gfCNCPoint3[21212] = {X 51.6286, Y 45.9257, Z -4.6667, A 0.000, B 0.000, C 0.000 }
gfCNCPoint3[21213] = {X 51.3210, Y 46.8050, Z -4.6667, A 0.000, B 0.000, C 0.000 }
gfCNCPoint3[21214] = {X 50.8253, Y 47.5937, Z -4.6667, A 0.000, B 0.000, C 0.000 }
gfCNCPoint3[21215] = {X 50.1666, Y 48.2524, Z -4.6667, A 0.000, B 0.000, C 0.000 }
gfCNCPoint3[21216] = {X 49.3779, Y 48.7480, Z -4.6667, A 0.000, B 0.000, C 0.000 }
gfCNCPoint3[21217] = {X 48.4986, Y 49.0557, Z -4.6667, A 0.000, B 0.000, C 0.000 }
gfCNCPoint3[21218] = {X 47.5729, Y 49.1600, Z -4.6667, A 0.000, B 0.000, C 0.000 }
gfCNCPoint3[21219] = {X 40.6393, Y 49.1600, Z -4.6667, A 0.000, B 0.000, C 0.000 }
gfCNCPoint3[21220] = {X 39.7136, Y 49.0557, Z -4.6667, A 0.000, B 0.000, C 0.000 }
gfCNCPoint3[21221] = {X 38.8343, Y 48.7480, Z -4.6667, A 0.000, B 0.000, C 0.000 }
gfCNCPoint3[21222] = {X 38.0456, Y 48.2524, Z -4.6667, A 0.000, B 0.000, C 0.000 }
gfCNCPoint3[21223] = {X 37.3869, Y 47.5937, Z -4.6667, A 0.000, B 0.000, C 0.000 }
gfCNCPoint3[21224] = {X 36.8913, Y 46.8050, Z -4.6667, A 0.000, B 0.000, C 0.000 }
gfCNCPoint3[21225] = {X 36.5836, Y 45.9257, Z -4.6667, A 0.000, B 0.000, C 0.000 }
gfCNCPoint3[21226] = {X 36.4793, Y 45.0000, Z -4.6667, A 0.000, B 0.000, C 0.000 }
gfCNCPoint3[21227] = {X 36.4793, Y 44.2086, Z -4.6667, A 0.000, B 0.000, C 0.000 }
gfCNCPoint3[21228] = {X 36.5946, Y 43.2363, Z -4.6667, A 0.000, B 0.000, C 0.000 }
gfCNCPoint3[21229] = {X 36.9339, Y 42.3179, Z -4.6667, A 0.000, B 0.000, C 0.000 }
gfCNCPoint3[21230] = {X 37.4785, Y 41.5042, Z -4.6667, A 0.000, B 0.000, C 0.000 }
gfCNCPoint3[21231] = {X 38.1981, Y 40.8404, Z -4.6667, A 0.000, B 0.000, C 0.000 }
gfCNCPoint3[21232] = {X 39.0530, Y 40.3631, Z -4.6667, A 0.000, B 0.000, C 0.000 }
gfCNCPoint3[21233] = {X 39.6600, Y 38.9340, Z -4.6667, A 0.000, B 0.000, C 0.000 }
gfCNCPoint3[21234] = {X 40.2148, Y 37.4838, Z -4.6667, A 0.000, B 0.000, C 0.000 }
gfCNCPoint3[21235] = {X 43.7983, Y 27.8629, Z -4.6667, A 0.000, B 0.000, C 0.000 }
gfCNCPoint3[21236] = {X 40.0498, Y 26.4668, Z -4.6667, A 0.000, B 0.000, C 0.000 }
gfCNCPoint3[21237] = {X 43.8732, Y 27.8908, Z -4.6667, A 0.000, B 0.000, C 0.000 }
gfCNCPoint3[21238] = {X 48.5582, Y 15.3126, Z -4.6667, A 0.000, B 0.000, C 0.000 }
gfCNCPoint3[21239] = {X 48.1610, Y 14.6012, Z -4.6667, A 0.000, B 0.000, C 0.000 }
gfCNCPoint3[21240] = {X 47.9131, Y 13.8250, Z -4.6667, A 0.000, B 0.000, C 0.000 }
gfCNCPoint3[21241] = {X 47.8244, Y 13.0150, Z -4.6667, A 0.000, B 0.000, C 0.000 }
gfCNCPoint3[21242] = {X 47.8242, Y 12.1868, Z -4.6667, A 0.000, B 0.000, C 0.000 }
gfCNCPoint3[21243] = {X 47.9265, Y 11.2789, Z -4.6667, A 0.000, B 0.000, C 0.000 }
gfCNCPoint3[21244] = {X 48.2283, Y 10.4166, Z -4.6667, A 0.000, B 0.000, C 0.000 }
gfCNCPoint3[21245] = {X 48.7144, Y 9.6430, Z -4.6667, A 0.000, B 0.000, C 0.000 }
gfCNCPoint3[21246] = {X 49.3604, Y 8.9969, Z -4.6667, A 0.000, B 0.000, C 0.000 }
gfCNCPoint3[21247] = {X 50.1340, Y 8.5109, Z -4.6667, A 0.000, B 0.000, C 0.000 }
gfCNCPoint3[21248] = {X 50.9963, Y 8.2091, Z -4.6667, A 0.000, B 0.000, C 0.000 }
gfCNCPoint3[21249] = {X 51.9042, Y 8.1068, Z -4.6667, A 0.000, B 0.000, C 0.000 }
gfCNCPoint3[21250] = {X 59.6221, Y 8.1068, Z -4.6667, A 0.000, B 0.000, C 0.000 }
gfCNCPoint3[21251] = {X 60.5300, Y 8.2091, Z -4.6667, A 0.000, B 0.000, C 0.000 }
gfCNCPoint3[21252] = {X 61.3924, Y 8.5109, Z -4.6667, A 0.000, B 0.000, C 0.000 }
gfCNCPoint3[21253] = {X 62.1660, Y 8.9969, Z -4.6667, A 0.000, B 0.000, C 0.000 }
gfCNCPoint3[21254] = {X 62.8120, Y 9.6430, Z -4.6667, A 0.000, B 0.000, C 0.000 }
gfCNCPoint3[21255] = {X 63.2981, Y 10.4166, Z -4.6667, A 0.000, B 0.000, C 0.000 }
gfCNCPoint3[21256] = {X 63.5998, Y 11.2789, Z -4.6667, A 0.000, B 0.000, C 0.000 }
gfCNCPoint3[21257] = {X 63.7021, Y 12.1868, Z -4.6667, A 0.000, B 0.000, C 0.000 }
gfCNCPoint3[21258] = {X 63.7021, Y 12.9781, Z -4.6667, A 0.000, B 0.000, C 0.000 }
gfCNCPoint3[21259] = {X 63.6148, Y 13.8177, Z -4.6667, A 0.000, B 0.000, C 0.000 }
gfCNCPoint3[21260] = {X 63.3566, Y 14.6213, Z -4.6667, A 0.000, B 0.000, C 0.000 }
gfCNCPoint3[21261] = {X 62.9385, Y 15.3546, Z -4.6667, A 0.000, B 0.000, C 0.000 }
gfCNCPoint3[21262] = {X 63.2013, Y 16.0481, Z -4.6667, A 0.000, B 0.000, C 0.000 }
gfCNCPoint3[21263] = {X 66.0153, Y 23.5152, Z -4.6667, A 0.000, B 0.000, C 0.000 }
gfCNCPoint3[21264] = {X 71.9857, Y 39.5865, Z -4.6667, A 0.000, B 0.000, C 0.000 }
gfCNCPoint3[21265] = {X 72.3285, Y 40.4488, Z -4.6667, A 0.000, B 0.000, C 0.000 }
gfCNCPoint3[21266] = {X 73.1525, Y 40.9152, Z -4.6667, A 0.000, B 0.000, C 0.000 }
gfCNCPoint3[21267] = {X 73.8468, Y 41.5589, Z -4.6667, A 0.000, B 0.000, C 0.000 }
gfCNCPoint3[21268] = {X 74.3740, Y 42.3453, Z -4.6667, A 0.000, B 0.000, C 0.000 }
gfCNCPoint3[21269] = {X 74.7058, Y 43.2320, Z -4.6667, A 0.000, B 0.000, C 0.000 }
gfCNCPoint3[21270] = {X 74.8243, Y 44.1714, Z -4.6667, A 0.000, B 0.000, C 0.000 }
gfCNCPoint3[21271] = {X 74.8245, Y 45.0000, Z -4.6667, A 0.000, B 0.000, C 0.000 }
gfCNCPoint3[21272] = {X 74.7222, Y 45.9079, Z -4.6667, A 0.000, B 0.000, C 0.000 }
gfCNCPoint3[21273] = {X 74.4204, Y 46.7702, Z -4.6667, A 0.000, B 0.000, C 0.000 }
gfCNCPoint3[21274] = {X 73.9343, Y 47.5438, Z -4.6667, A 0.000, B 0.000, C 0.000 }
gfCNCPoint3[21275] = {X 73.2883, Y 48.1899, Z -4.6667, A 0.000, B 0.000, C 0.000 }
gfCNCPoint3[21276] = {X 72.5147, Y 48.6760, Z -4.6667, A 0.000, B 0.000, C 0.000 }
gfCNCPoint3[21277] = {X 71.6523, Y 48.9777, Z -4.6667, A 0.000, B 0.000, C 0.000 }
gfCNCPoint3[21278] = {X 70.7445, Y 49.0800, Z -4.6667, A 0.000, B 0.000, C 0.000 }
gfCNCPoint3[21279] = {X 64.1851, Y 49.0800, Z -4.6667, A 0.000, B 0.000, C 0.000 }
gfCNCPoint3[21280] = {X 63.2772, Y 48.9777, Z -4.6667, A 0.000, B 0.000, C 0.000 }
gfCNCPoint3[21281] = {X 62.4149, Y 48.6760, Z -4.6667, A 0.000, B 0.000, C 0.000 }
gfCNCPoint3[21282] = {X 61.6413, Y 48.1899, Z -4.6667, A 0.000, B 0.000, C 0.000 }
gfCNCPoint3[21283] = {X 60.9953, Y 47.5438, Z -4.6667, A 0.000, B 0.000, C 0.000 }
gfCNCPoint3[21284] = {X 60.5092, Y 46.7702, Z -4.6667, A 0.000, B 0.000, C 0.000 }
gfCNCPoint3[21285] = {X 60.2074, Y 45.9079, Z -4.6667, A 0.000, B 0.000, C 0.000 }
gfCNCPoint3[21286] = {X 60.1051, Y 45.0000, Z -4.6667, A 0.000, B 0.000, C 0.000 }
gfCNCPoint3[21287] = {X 60.1051, Y 44.2086, Z -4.6667, A 0.000, B 0.000, C 0.000 }
gfCNCPoint3[21288] = {X 60.1954, Y 43.3580, Z -4.6667, A 0.000, B 0.000, C 0.000 }
gfCNCPoint3[21289] = {X 60.4610, Y 42.5449, Z -4.6667, A 0.000, B 0.000, C 0.000 }
gfCNCPoint3[21290] = {X 60.8902, Y 41.8051, Z -4.6667, A 0.000, B 0.000, C 0.000 }
gfCNCPoint3[21291] = {X 60.1747, Y 39.8492, Z -4.6667, A 0.000, B 0.000, C 0.000 }
gfCNCPoint3[21292] = {X 51.9106, Y 39.8492, Z -4.6667, A 0.000, B 0.000, C 0.000 }
gfCNCPoint3[21293] = {X 51.0693, Y 42.1093, Z -4.6667, A 0.000, B 0.000, C 0.000 }
gfCNCPoint3[21294] = {X 51.1301, Y 42.2105, Z -4.6667, A 0.000, B 0.000, C 0.000 }
gfCNCPoint3[21295] = {X 51.4138, Y 42.8325, Z -4.6667, A 0.000, B 0.000, C 0.000 }
gfCNCPoint3[21296] = {X 51.5897, Y 43.4932, Z -4.6667, A 0.000, B 0.000, C 0.000 }
gfCNCPoint3[21297] = {X 51.6528, Y 44.1740, Z -4.6667, A 0.000, B 0.000, C 0.000 }
gfCNCPoint3[21298] = {X 51.6529, Y 45.0000, Z -4.6667, A 0.000, B 0.000, C 0.000 }
gfCNCPoint3[21299] = {X 51.5506, Y 45.9079, Z -4.6667, A 0.000, B 0.000, C 0.000 }
gfCNCPoint3[21300] = {X 51.2489, Y 46.7702, Z -4.6667, A 0.000, B 0.000, C 0.000 }
gfCNCPoint3[21301] = {X 50.7628, Y 47.5438, Z -4.6667, A 0.000, B 0.000, C 0.000 }
gfCNCPoint3[21302] = {X 50.1168, Y 48.1899, Z -4.6667, A 0.000, B 0.000, C 0.000 }
gfCNCPoint3[21303] = {X 49.3432, Y 48.6760, Z -4.6667, A 0.000, B 0.000, C 0.000 }
gfCNCPoint3[21304] = {X 48.4808, Y 48.9777, Z -4.6667, A 0.000, B 0.000, C 0.000 }
gfCNCPoint3[21305] = {X 47.5729, Y 49.0800, Z -4.6667, A 0.000, B 0.000, C 0.000 }
gfCNCPoint3[21306] = {X 40.6393, Y 49.0800, Z -4.6667, A 0.000, B 0.000, C 0.000 }
gfCNCPoint3[21307] = {X 39.7314, Y 48.9777, Z -4.6667, A 0.000, B 0.000, C 0.000 }
gfCNCPoint3[21308] = {X 38.8691, Y 48.6760, Z -4.6667, A 0.000, B 0.000, C 0.000 }
gfCNCPoint3[21309] = {X 38.0955, Y 48.1899, Z -4.6667, A 0.000, B 0.000, C 0.000 }
gfCNCPoint3[21310] = {X 37.4494, Y 47.5438, Z -4.6667, A 0.000, B 0.000, C 0.000 }
gfCNCPoint3[21311] = {X 36.9633, Y 46.7702, Z -4.6667, A 0.000, B 0.000, C 0.000 }
gfCNCPoint3[21312] = {X 36.6616, Y 45.9079, Z -4.6667, A 0.000, B 0.000, C 0.000 }
gfCNCPoint3[21313] = {X 36.5593, Y 45.0000, Z -4.6667, A 0.000, B 0.000, C 0.000 }
gfCNCPoint3[21314] = {X 36.5593, Y 44.2086, Z -4.6667, A 0.000, B 0.000, C 0.000 }
gfCNCPoint3[21315] = {X 36.6736, Y 43.2499, Z -4.6667, A 0.000, B 0.000, C 0.000 }
gfCNCPoint3[21316] = {X 37.0099, Y 42.3449, Z -4.6667, A 0.000, B 0.000, C 0.000 }
gfCNCPoint3[21317] = {X 37.5495, Y 41.5443, Z -4.6667, A 0.000, B 0.000, C 0.000 }
gfCNCPoint3[21318] = {X 38.2621, Y 40.8928, Z -4.6667, A 0.000, B 0.000, C 0.000 }
gfCNCPoint3[21319] = {X 39.1079, Y 40.4271, Z -4.6667, A 0.000, B 0.000, C 0.000 }
gfCNCPoint3[21320] = {X 39.1261, Y 40.3957, Z -4.6667, A 0.000, B 0.000, C 0.000 }
gfCNCPoint3[21321] = {X 39.7342, Y 38.9639, Z -4.6667, A 0.000, B 0.000, C 0.000 }
gfCNCPoint3[21322] = {X 40.2900, Y 37.5111, Z -4.6667, A 0.000, B 0.000, C 0.000 }
gfCNCPoint3[21323] = {X 43.8732, Y 27.8908, Z -4.6667, A 0.000, B 0.000, C 0.000 }
gfCNCPoint3[21324] = {X 40.1248, Y 26.4947, Z -4.6667, A 0.000, B 0.000, C 0.000 }
gfCNCPoint3[21325] = {X 43.9482, Y 27.9188, Z -4.6667, A 0.000, B 0.000, C 0.000 }
gfCNCPoint3[21326] = {X 48.6479, Y 15.3010, Z -4.6667, A 0.000, B 0.000, C 0.000 }
gfCNCPoint3[21327] = {X 48.2407, Y 14.5838, Z -4.6667, A 0.000, B 0.000, C 0.000 }
gfCNCPoint3[21328] = {X 47.9892, Y 13.7983, Z -4.6667, A 0.000, B 0.000, C 0.000 }
gfCNCPoint3[21329] = {X 47.9042, Y 12.9779, Z -4.6667, A 0.000, B 0.000, C 0.000 }
gfCNCPoint3[21330] = {X 47.9042, Y 12.1868, Z -4.6667, A 0.000, B 0.000, C 0.000 }
gfCNCPoint3[21331] = {X 48.0045, Y 11.2967, Z -4.6667, A 0.000, B 0.000, C 0.000 }
gfCNCPoint3[21332] = {X 48.3003, Y 10.4513, Z -4.6667, A 0.000, B 0.000, C 0.000 }
gfCNCPoint3[21333] = {X 48.7769, Y 9.6929, Z -4.6667, A 0.000, B 0.000, C 0.000 }
gfCNCPoint3[21334] = {X 49.4103, Y 9.0595, Z -4.6667, A 0.000, B 0.000, C 0.000 }
gfCNCPoint3[21335] = {X 50.1687, Y 8.5829, Z -4.6667, A 0.000, B 0.000, C 0.000 }
gfCNCPoint3[21336] = {X 51.0141, Y 8.2871, Z -4.6667, A 0.000, B 0.000, C 0.000 }
gfCNCPoint3[21337] = {X 51.9042, Y 8.1868, Z -4.6667, A 0.000, B 0.000, C 0.000 }
gfCNCPoint3[21338] = {X 59.6221, Y 8.1868, Z -4.6667, A 0.000, B 0.000, C 0.000 }
gfCNCPoint3[21339] = {X 60.5122, Y 8.2871, Z -4.6667, A 0.000, B 0.000, C 0.000 }
gfCNCPoint3[21340] = {X 61.3577, Y 8.5829, Z -4.6667, A 0.000, B 0.000, C 0.000 }
gfCNCPoint3[21341] = {X 62.1161, Y 9.0595, Z -4.6667, A 0.000, B 0.000, C 0.000 }
gfCNCPoint3[21342] = {X 62.7495, Y 9.6929, Z -4.6667, A 0.000, B 0.000, C 0.000 }
gfCNCPoint3[21343] = {X 63.2260, Y 10.4513, Z -4.6667, A 0.000, B 0.000, C 0.000 }
gfCNCPoint3[21344] = {X 63.5218, Y 11.2967, Z -4.6667, A 0.000, B 0.000, C 0.000 }
gfCNCPoint3[21345] = {X 63.6221, Y 12.1868, Z -4.6667, A 0.000, B 0.000, C 0.000 }
gfCNCPoint3[21346] = {X 63.6219, Y 13.0192, Z -4.6667, A 0.000, B 0.000, C 0.000 }
gfCNCPoint3[21347] = {X 63.5277, Y 13.8419, Z -4.6667, A 0.000, B 0.000, C 0.000 }
gfCNCPoint3[21348] = {X 63.2661, Y 14.6276, Z -4.6667, A 0.000, B 0.000, C 0.000 }
gfCNCPoint3[21349] = {X 62.8484, Y 15.3426, Z -4.6667, A 0.000, B 0.000, C 0.000 }
gfCNCPoint3[21350] = {X 63.1264, Y 16.0764, Z -4.6667, A 0.000, B 0.000, C 0.000 }
gfCNCPoint3[21351] = {X 65.9404, Y 23.5433, Z -4.6667, A 0.000, B 0.000, C 0.000 }
gfCNCPoint3[21352] = {X 71.9110, Y 39.6152, Z -4.6667, A 0.000, B 0.000, C 0.000 }
gfCNCPoint3[21353] = {X 72.2612, Y 40.4962, Z -4.6667, A 0.000, B 0.000, C 0.000 }
gfCNCPoint3[21354] = {X 72.2800, Y 40.5152, Z -4.6667, A 0.000, B 0.000, C 0.000 }
gfCNCPoint3[21355] = {X 72.3456, Y 40.5432, Z -4.6667, A 0.000, B 0.000, C 0.000 }
gfCNCPoint3[21356] = {X 72.4108, Y 40.5724, Z -4.6667, A 0.000, B 0.000, C 0.000 }
gfCNCPoint3[21357] = {X 73.1903, Y 41.0437, Z -4.6667, A 0.000, B 0.000, C 0.000 }
gfCNCPoint3[21358] = {X 73.8430, Y 41.6791, Z -4.6667, A 0.000, B 0.000, C 0.000 }
gfCNCPoint3[21359] = {X 74.3350, Y 42.4458, Z -4.6667, A 0.000, B 0.000, C 0.000 }
gfCNCPoint3[21360] = {X 74.6408, Y 43.3039, Z -4.6667, A 0.000, B 0.000, C 0.000 }
gfCNCPoint3[21361] = {X 74.7445, Y 44.2089, Z -4.6667, A 0.000, B 0.000, C 0.000 }
gfCNCPoint3[21362] = {X 74.7445, Y 45.0000, Z -4.6667, A 0.000, B 0.000, C 0.000 }
gfCNCPoint3[21363] = {X 74.6442, Y 45.8901, Z -4.6667, A 0.000, B 0.000, C 0.000 }
gfCNCPoint3[21364] = {X 74.3483, Y 46.7355, Z -4.6667, A 0.000, B 0.000, C 0.000 }
gfCNCPoint3[21365] = {X 73.8718, Y 47.4940, Z -4.6667, A 0.000, B 0.000, C 0.000 }
gfCNCPoint3[21366] = {X 73.2384, Y 48.1273, Z -4.6667, A 0.000, B 0.000, C 0.000 }
gfCNCPoint3[21367] = {X 72.4800, Y 48.6039, Z -4.6667, A 0.000, B 0.000, C 0.000 }
gfCNCPoint3[21368] = {X 71.6345, Y 48.8997, Z -4.6667, A 0.000, B 0.000, C 0.000 }
gfCNCPoint3[21369] = {X 70.7445, Y 49.0000, Z -4.6667, A 0.000, B 0.000, C 0.000 }
gfCNCPoint3[21370] = {X 64.1851, Y 49.0000, Z -4.6667, A 0.000, B 0.000, C 0.000 }
gfCNCPoint3[21371] = {X 63.2951, Y 48.8997, Z -4.6667, A 0.000, B 0.000, C 0.000 }
gfCNCPoint3[21372] = {X 62.4496, Y 48.6039, Z -4.6667, A 0.000, B 0.000, C 0.000 }
gfCNCPoint3[21373] = {X 61.6912, Y 48.1273, Z -4.6667, A 0.000, B 0.000, C 0.000 }
gfCNCPoint3[21374] = {X 61.0578, Y 47.4940, Z -4.6667, A 0.000, B 0.000, C 0.000 }
gfCNCPoint3[21375] = {X 60.5813, Y 46.7355, Z -4.6667, A 0.000, B 0.000, C 0.000 }
gfCNCPoint3[21376] = {X 60.2854, Y 45.8901, Z -4.6667, A 0.000, B 0.000, C 0.000 }
gfCNCPoint3[21377] = {X 60.1851, Y 45.0000, Z -4.6667, A 0.000, B 0.000, C 0.000 }
gfCNCPoint3[21378] = {X 60.1855, Y 44.1538, Z -4.6667, A 0.000, B 0.000, C 0.000 }
gfCNCPoint3[21379] = {X 60.2746, Y 43.3674, Z -4.6667, A 0.000, B 0.000, C 0.000 }
gfCNCPoint3[21380] = {X 60.5168, Y 42.6140, Z -4.6667, A 0.000, B 0.000, C 0.000 }
gfCNCPoint3[21381] = {X 60.9025, Y 41.9231, Z -4.6667, A 0.000, B 0.000, C 0.000 }
gfCNCPoint3[21382] = {X 60.9801, Y 41.8180, Z -4.6667, A 0.000, B 0.000, C 0.000 }
gfCNCPoint3[21383] = {X 60.2306, Y 39.7692, Z -4.6667, A 0.000, B 0.000, C 0.000 }
gfCNCPoint3[21384] = {X 51.8424, Y 39.7692, Z -4.6667, A 0.000, B 0.000, C 0.000 }
gfCNCPoint3[21385] = {X 51.8424, Y 39.8029, Z -4.6667, A 0.000, B 0.000, C 0.000 }
gfCNCPoint3[21386] = {X 50.9809, Y 42.1174, Z -4.6667, A 0.000, B 0.000, C 0.000 }
gfCNCPoint3[21387] = {X 51.0725, Y 42.2716, Z -4.6667, A 0.000, B 0.000, C 0.000 }
gfCNCPoint3[21388] = {X 51.3479, Y 42.8860, Z -4.6667, A 0.000, B 0.000, C 0.000 }
gfCNCPoint3[21389] = {X 51.5163, Y 43.5380, Z -4.6667, A 0.000, B 0.000, C 0.000 }
gfCNCPoint3[21390] = {X 51.5729, Y 44.2089, Z -4.6667, A 0.000, B 0.000, C 0.000 }
gfCNCPoint3[21391] = {X 51.5729, Y 45.0000, Z -4.6667, A 0.000, B 0.000, C 0.000 }
gfCNCPoint3[21392] = {X 51.4726, Y 45.8901, Z -4.6667, A 0.000, B 0.000, C 0.000 }
gfCNCPoint3[21393] = {X 51.1768, Y 46.7355, Z -4.6667, A 0.000, B 0.000, C 0.000 }
gfCNCPoint3[21394] = {X 50.7003, Y 47.4940, Z -4.6667, A 0.000, B 0.000, C 0.000 }
gfCNCPoint3[21395] = {X 50.0669, Y 48.1273, Z -4.6667, A 0.000, B 0.000, C 0.000 }
gfCNCPoint3[21396] = {X 49.3085, Y 48.6039, Z -4.6667, A 0.000, B 0.000, C 0.000 }
gfCNCPoint3[21397] = {X 48.4630, Y 48.8997, Z -4.6667, A 0.000, B 0.000, C 0.000 }
gfCNCPoint3[21398] = {X 47.5729, Y 49.0000, Z -4.6667, A 0.000, B 0.000, C 0.000 }
gfCNCPoint3[21399] = {X 40.6393, Y 49.0000, Z -4.6667, A 0.000, B 0.000, C 0.000 }
gfCNCPoint3[21400] = {X 39.7492, Y 48.8997, Z -4.6667, A 0.000, B 0.000, C 0.000 }
gfCNCPoint3[21401] = {X 38.9038, Y 48.6039, Z -4.6667, A 0.000, B 0.000, C 0.000 }
gfCNCPoint3[21402] = {X 38.1453, Y 48.1273, Z -4.6667, A 0.000, B 0.000, C 0.000 }
gfCNCPoint3[21403] = {X 37.5120, Y 47.4940, Z -4.6667, A 0.000, B 0.000, C 0.000 }
gfCNCPoint3[21404] = {X 37.0354, Y 46.7355, Z -4.6667, A 0.000, B 0.000, C 0.000 }
gfCNCPoint3[21405] = {X 36.7396, Y 45.8901, Z -4.6667, A 0.000, B 0.000, C 0.000 }
gfCNCPoint3[21406] = {X 36.6393, Y 45.0000, Z -4.6667, A 0.000, B 0.000, C 0.000 }
gfCNCPoint3[21407] = {X 36.6397, Y 44.1538, Z -4.6667, A 0.000, B 0.000, C 0.000 }
gfCNCPoint3[21408] = {X 36.7563, Y 43.2482, Z -4.6667, A 0.000, B 0.000, C 0.000 }
gfCNCPoint3[21409] = {X 37.0753, Y 42.3928, Z -4.6667, A 0.000, B 0.000, C 0.000 }
gfCNCPoint3[21410] = {X 37.5799, Y 41.6319, Z -4.6667, A 0.000, B 0.000, C 0.000 }
gfCNCPoint3[21411] = {X 38.2440, Y 41.0053, Z -4.6667, A 0.000, B 0.000, C 0.000 }
gfCNCPoint3[21412] = {X 39.0328, Y 40.5456, Z -4.6667, A 0.000, B 0.000, C 0.000 }
gfCNCPoint3[21413] = {X 39.0852, Y 40.5230, Z -4.6667, A 0.000, B 0.000, C 0.000 }
gfCNCPoint3[21414] = {X 39.1379, Y 40.5013, Z -4.6667, A 0.000, B 0.000, C 0.000 }
gfCNCPoint3[21415] = {X 39.1678, Y 40.4818, Z -4.6667, A 0.000, B 0.000, C 0.000 }
gfCNCPoint3[21416] = {X 39.1882, Y 40.4527, Z -4.6667, A 0.000, B 0.000, C 0.000 }
gfCNCPoint3[21417] = {X 39.2130, Y 40.3971, Z -4.6667, A 0.000, B 0.000, C 0.000 }
gfCNCPoint3[21418] = {X 39.2378, Y 40.3415, Z -4.6667, A 0.000, B 0.000, C 0.000 }
gfCNCPoint3[21419] = {X 39.8262, Y 38.9498, Z -4.6667, A 0.000, B 0.000, C 0.000 }
gfCNCPoint3[21420] = {X 40.3652, Y 37.5383, Z -4.6667, A 0.000, B 0.000, C 0.000 }
gfCNCPoint3[21421] = {X 43.9482, Y 27.9188, Z -4.6667, A 0.000, B 0.000, C 0.000 }
gfCNCPoint3[21422] = {X 40.1248, Y 26.4947, Z -4.6667, A 0.000, B 0.000, C 0.000 }
gfCNCPoint3[21423] = {X 40.1248, Y 26.4947, Z -1.6667, A 0.000, B 0.000, C 0.000 }
gfCNCPoint3[21424] = {X 40.1248, Y 26.4947, Z 11.0000, A 0.000, B 0.000, C 0.000 }
gfCNCPoint3[21425] = {X 79.0226, Y 28.5916, Z 11.0000, A 0.000, B 0.000, C 0.000 }
gfCNCPoint3[21426] = {X 79.0226, Y 28.5916, Z -1.6667, A 0.000, B 0.000, C 0.000 }
gfCNCPoint3[21427] = {X 79.0226, Y 28.5916, Z -4.6667, A 0.000, B 0.000, C 0.000 }
gfCNCPoint3[21428] = {X 83.1026, Y 28.5916, Z -4.6667, A 0.000, B 0.000, C 0.000 }
gfCNCPoint3[21429] = {X 83.1025, Y 16.2741, Z -4.6667, A 0.000, B 0.000, C 0.000 }
gfCNCPoint3[21430] = {X 82.4640, Y 15.6030, Z -4.6667, A 0.000, B 0.000, C 0.000 }
gfCNCPoint3[21431] = {X 81.9833, Y 14.8112, Z -4.6667, A 0.000, B 0.000, C 0.000 }
gfCNCPoint3[21432] = {X 81.6824, Y 13.9351, Z -4.6667, A 0.000, B 0.000, C 0.000 }
gfCNCPoint3[21433] = {X 81.5752, Y 13.0150, Z -4.6667, A 0.000, B 0.000, C 0.000 }
gfCNCPoint3[21434] = {X 81.5751, Y 12.1868, Z -4.6667, A 0.000, B 0.000, C 0.000 }
gfCNCPoint3[21435] = {X 81.6834, Y 11.2255, Z -4.6667, A 0.000, B 0.000, C 0.000 }
gfCNCPoint3[21436] = {X 82.0029, Y 10.3125, Z -4.6667, A 0.000, B 0.000, C 0.000 }
gfCNCPoint3[21437] = {X 82.5176, Y 9.4933, Z -4.6667, A 0.000, B 0.000, C 0.000 }
gfCNCPoint3[21438] = {X 83.2016, Y 8.8093, Z -4.6667, A 0.000, B 0.000, C 0.000 }
gfCNCPoint3[21439] = {X 84.0207, Y 8.2946, Z -4.6667, A 0.000, B 0.000, C 0.000 }
gfCNCPoint3[21440] = {X 84.9338, Y 7.9751, Z -4.6667, A 0.000, B 0.000, C 0.000 }
gfCNCPoint3[21441] = {X 85.8951, Y 7.8668, Z -4.6667, A 0.000, B 0.000, C 0.000 }
gfCNCPoint3[21442] = {X 94.0497, Y 7.8668, Z -4.6667, A 0.000, B 0.000, C 0.000 }
gfCNCPoint3[21443] = {X 95.0110, Y 7.9751, Z -4.6667, A 0.000, B 0.000, C 0.000 }
gfCNCPoint3[21444] = {X 95.9240, Y 8.2946, Z -4.6667, A 0.000, B 0.000, C 0.000 }
gfCNCPoint3[21445] = {X 96.7431, Y 8.8093, Z -4.6667, A 0.000, B 0.000, C 0.000 }
gfCNCPoint3[21446] = {X 97.4272, Y 9.4933, Z -4.6667, A 0.000, B 0.000, C 0.000 }
gfCNCPoint3[21447] = {X 97.9419, Y 10.3124, Z -4.6667, A 0.000, B 0.000, C 0.000 }
gfCNCPoint3[21448] = {X 98.2614, Y 11.2255, Z -4.6667, A 0.000, B 0.000, C 0.000 }
gfCNCPoint3[21449] = {X 98.3697, Y 12.1868, Z -4.6667, A 0.000, B 0.000, C 0.000 }
gfCNCPoint3[21450] = {X 98.3697, Y 12.9782, Z -4.6667, A 0.000, B 0.000, C 0.000 }
gfCNCPoint3[21451] = {X 98.2967, Y 13.7680, Z -4.6667, A 0.000, B 0.000, C 0.000 }
gfCNCPoint3[21452] = {X 98.0805, Y 14.5312, Z -4.6667, A 0.000, B 0.000, C 0.000 }
gfCNCPoint3[21453] = {X 97.7285, Y 15.2420, Z -4.6667, A 0.000, B 0.000, C 0.000 }
gfCNCPoint3[21454] = {X 101.8778, Y 25.5286, Z -4.6667, A 0.000, B 0.000, C 0.000 }
gfCNCPoint3[21455] = {X 106.0165, Y 15.2214, Z -4.6667, A 0.000, B 0.000, C 0.000 }
gfCNCPoint3[21456] = {X 105.6761, Y 14.5285, Z -4.6667, A 0.000, B 0.000, C 0.000 }
gfCNCPoint3[21457] = {X 105.4645, Y 13.7861, Z -4.6667, A 0.000, B 0.000, C 0.000 }
gfCNCPoint3[21458] = {X 105.3885, Y 13.0179, Z -4.6667, A 0.000, B 0.000, C 0.000 }
gfCNCPoint3[21459] = {X 105.3883, Y 12.1868, Z -4.6667, A 0.000, B 0.000, C 0.000 }
gfCNCPoint3[21460] = {X 105.4966, Y 11.2255, Z -4.6667, A 0.000, B 0.000, C 0.000 }
gfCNCPoint3[21461] = {X 105.8161, Y 10.3124, Z -4.6667, A 0.000, B 0.000, C 0.000 }
gfCNCPoint3[21462] = {X 106.3308, Y 9.4933, Z -4.6667, A 0.000, B 0.000, C 0.000 }
gfCNCPoint3[21463] = {X 107.0148, Y 8.8093, Z -4.6667, A 0.000, B 0.000, C 0.000 }
gfCNCPoint3[21464] = {X 107.8339, Y 8.2946, Z -4.6667, A 0.000, B 0.000, C 0.000 }
gfCNCPoint3[21465] = {X 108.7470, Y 7.9751, Z -4.6667, A 0.000, B 0.000, C 0.000 }
gfCNCPoint3[21466] = {X 109.7083, Y 7.8668, Z -4.6667, A 0.000, B 0.000, C 0.000 }
gfCNCPoint3[21467] = {X 117.7916, Y 7.8668, Z -4.6667, A 0.000, B 0.000, C 0.000 }
gfCNCPoint3[21468] = {X 118.7529, Y 7.9751, Z -4.6667, A 0.000, B 0.000, C 0.000 }
gfCNCPoint3[21469] = {X 119.6660, Y 8.2946, Z -4.6667, A 0.000, B 0.000, C 0.000 }
gfCNCPoint3[21470] = {X 120.4851, Y 8.8093, Z -4.6667, A 0.000, B 0.000, C 0.000 }
gfCNCPoint3[21471] = {X 121.1691, Y 9.4933, Z -4.6667, A 0.000, B 0.000, C 0.000 }
gfCNCPoint3[21472] = {X 121.6838, Y 10.3124, Z -4.6667, A 0.000, B 0.000, C 0.000 }
gfCNCPoint3[21473] = {X 122.0033, Y 11.2255, Z -4.6667, A 0.000, B 0.000, C 0.000 }
gfCNCPoint3[21474] = {X 122.1116, Y 12.1868, Z -4.6667, A 0.000, B 0.000, C 0.000 }
gfCNCPoint3[21475] = {X 122.1116, Y 12.9782, Z -4.6667, A 0.000, B 0.000, C 0.000 }
gfCNCPoint3[21476] = {X 122.0103, Y 13.9078, Z -4.6667, A 0.000, B 0.000, C 0.000 }
gfCNCPoint3[21477] = {X 121.7114, Y 14.7939, Z -4.6667, A 0.000, B 0.000, C 0.000 }
gfCNCPoint3[21478] = {X 121.2288, Y 15.5949, Z -4.6667, A 0.000, B 0.000, C 0.000 }
gfCNCPoint3[21479] = {X 120.5851, Y 16.2732, Z -4.6667, A 0.000, B 0.000, C 0.000 }
gfCNCPoint3[21480] = {X 120.5841, Y 40.9142, Z -4.6667, A 0.000, B 0.000, C 0.000 }
gfCNCPoint3[21481] = {X 120.6222, Y 40.9454, Z -4.6667, A 0.000, B 0.000, C 0.000 }
gfCNCPoint3[21482] = {X 121.2456, Y 41.6142, Z -4.6667, A 0.000, B 0.000, C 0.000 }
gfCNCPoint3[21483] = {X 121.7143, Y 42.3991, Z -4.6667, A 0.000, B 0.000, C 0.000 }
gfCNCPoint3[21484] = {X 122.0072, Y 43.2651, Z -4.6667, A 0.000, B 0.000, C 0.000 }
gfCNCPoint3[21485] = {X 122.1114, Y 44.1734, Z -4.6667, A 0.000, B 0.000, C 0.000 }
gfCNCPoint3[21486] = {X 122.1116, Y 45.0000, Z -4.6667, A 0.000, B 0.000, C 0.000 }
gfCNCPoint3[21487] = {X 122.0033, Y 45.9613, Z -4.6667, A 0.000, B 0.000, C 0.000 }
gfCNCPoint3[21488] = {X 121.6838, Y 46.8744, Z -4.6667, A 0.000, B 0.000, C 0.000 }
gfCNCPoint3[21489] = {X 121.1691, Y 47.6935, Z -4.6667, A 0.000, B 0.000, C 0.000 }
gfCNCPoint3[21490] = {X 120.4851, Y 48.3775, Z -4.6667, A 0.000, B 0.000, C 0.000 }
gfCNCPoint3[21491] = {X 119.6660, Y 48.8922, Z -4.6667, A 0.000, B 0.000, C 0.000 }
gfCNCPoint3[21492] = {X 118.7529, Y 49.2117, Z -4.6667, A 0.000, B 0.000, C 0.000 }
gfCNCPoint3[21493] = {X 117.7916, Y 49.3200, Z -4.6667, A 0.000, B 0.000, C 0.000 }
gfCNCPoint3[21494] = {X 111.9185, Y 49.3200, Z -4.6667, A 0.000, B 0.000, C 0.000 }
gfCNCPoint3[21495] = {X 110.9619, Y 49.2128, Z -4.6667, A 0.000, B 0.000, C 0.000 }
gfCNCPoint3[21496] = {X 110.0529, Y 48.8964, Z -4.6667, A 0.000, B 0.000, C 0.000 }
gfCNCPoint3[21497] = {X 109.2365, Y 48.3866, Z -4.6667, A 0.000, B 0.000, C 0.000 }
gfCNCPoint3[21498] = {X 108.5532, Y 47.7087, Z -4.6667, A 0.000, B 0.000, C 0.000 }
gfCNCPoint3[21499] = {X 108.0369, Y 46.8963, Z -4.6667, A 0.000, B 0.000, C 0.000 }
gfCNCPoint3[21500] = {X 107.7134, Y 45.9898, Z -4.6667, A 0.000, B 0.000, C 0.000 }
gfCNCPoint3[21501] = {X 107.5986, Y 45.0341, Z -4.6667, A 0.000, B 0.000, C 0.000 }
gfCNCPoint3[21502] = {X 107.5985, Y 44.1775, Z -4.6667, A 0.000, B 0.000, C 0.000 }
gfCNCPoint3[21503] = {X 107.6340, Y 43.6361, Z -4.6667, A 0.000, B 0.000, C 0.000 }
gfCNCPoint3[21504] = {X 107.7398, Y 43.1039, Z -4.6667, A 0.000, B 0.000, C 0.000 }
gfCNCPoint3[21505] = {X 107.9075, Y 42.6066, Z -4.6667, A 0.000, B 0.000, C 0.000 }
gfCNCPoint3[21506] = {X 108.1365, Y 42.1345, Z -4.6667, A 0.000, B 0.000, C 0.000 }
gfCNCPoint3[21507] = {X 108.5869, Y 41.4639, Z -4.6667, A 0.000, B 0.000, C 0.000 }
gfCNCPoint3[21508] = {X 109.1259, Y 40.8623, Z -4.6667, A 0.000, B 0.000, C 0.000 }
gfCNCPoint3[21509] = {X 109.1258, Y 39.2961, Z -4.6667, A 0.000, B 0.000, C 0.000 }
gfCNCPoint3[21510] = {X 106.1118, Y 46.6615, Z -4.6667, A 0.000, B 0.000, C 0.000 }
gfCNCPoint3[21511] = {X 105.7417, Y 47.3611, Z -4.6667, A 0.000, B 0.000, C 0.000 }
gfCNCPoint3[21512] = {X 105.2502, Y 47.9815, Z -4.6667, A 0.000, B 0.000, C 0.000 }
gfCNCPoint3[21513] = {X 104.6538, Y 48.5018, Z -4.6667, A 0.000, B 0.000, C 0.000 }
gfCNCPoint3[21514] = {X 103.9724, Y 48.9046, Z -4.6667, A 0.000, B 0.000, C 0.000 }
gfCNCPoint3[21515] = {X 103.0287, Y 49.2242, Z -4.6667, A 0.000, B 0.000, C 0.000 }
gfCNCPoint3[21516] = {X 102.0368, Y 49.3191, Z -4.6667, A 0.000, B 0.000, C 0.000 }
gfCNCPoint3[21517] = {X 101.0496, Y 49.1842, Z -4.6667, A 0.000, B 0.000, C 0.000 }
gfCNCPoint3[21518] = {X 100.1195, Y 48.8268, Z -4.6667, A 0.000, B 0.000, C 0.000 }
gfCNCPoint3[21519] = {X 99.2961, Y 48.2657, Z -4.6667, A 0.000, B 0.000, C 0.000 }
gfCNCPoint3[21520] = {X 98.6231, Y 47.5309, Z -4.6667, A 0.000, B 0.000, C 0.000 }
gfCNCPoint3[21521] = {X 98.1363, Y 46.6615, Z -4.6667, A 0.000, B 0.000, C 0.000 }
gfCNCPoint3[21522] = {X 95.1310, Y 39.3117, Z -4.6667, A 0.000, B 0.000, C 0.000 }
gfCNCPoint3[21523] = {X 95.1311, Y 40.9051, Z -4.6667, A 0.000, B 0.000, C 0.000 }
gfCNCPoint3[21524] = {X 95.6585, Y 41.4454, Z -4.6667, A 0.000, B 0.000, C 0.000 }
gfCNCPoint3[21525] = {X 96.0858, Y 42.0679, Z -4.6667, A 0.000, B 0.000, C 0.000 }
gfCNCPoint3[21526] = {X 96.3311, Y 42.5731, Z -4.6667, A 0.000, B 0.000, C 0.000 }
gfCNCPoint3[21527] = {X 96.5101, Y 43.1054, Z -4.6667, A 0.000, B 0.000, C 0.000 }
gfCNCPoint3[21528] = {X 96.6192, Y 43.6512, Z -4.6667, A 0.000, B 0.000, C 0.000 }
gfCNCPoint3[21529] = {X 96.6585, Y 44.2065, Z -4.6667, A 0.000, B 0.000, C 0.000 }
gfCNCPoint3[21530] = {X 96.6583, Y 45.0415, Z -4.6667, A 0.000, B 0.000, C 0.000 }
gfCNCPoint3[21531] = {X 96.5422, Y 45.9960, Z -4.6667, A 0.000, B 0.000, C 0.000 }
gfCNCPoint3[21532] = {X 96.2178, Y 46.9011, Z -4.6667, A 0.000, B 0.000, C 0.000 }
gfCNCPoint3[21533] = {X 95.7012, Y 47.7120, Z -4.6667, A 0.000, B 0.000, C 0.000 }
gfCNCPoint3[21534] = {X 95.0181, Y 48.3886, Z -4.6667, A 0.000, B 0.000, C 0.000 }
gfCNCPoint3[21535] = {X 94.2022, Y 48.8973, Z -4.6667, A 0.000, B 0.000, C 0.000 }
gfCNCPoint3[21536] = {X 93.2940, Y 49.2130, Z -4.6667, A 0.000, B 0.000, C 0.000 }
gfCNCPoint3[21537] = {X 92.3385, Y 49.3200, Z -4.6667, A 0.000, B 0.000, C 0.000 }
gfCNCPoint3[21538] = {X 85.8951, Y 49.3200, Z -4.6667, A 0.000, B 0.000, C 0.000 }
gfCNCPoint3[21539] = {X 84.9387, Y 49.2128, Z -4.6667, A 0.000, B 0.000, C 0.000 }
gfCNCPoint3[21540] = {X 84.0297, Y 48.8965, Z -4.6667, A 0.000, B 0.000, C 0.000 }
gfCNCPoint3[21541] = {X 83.2134, Y 48.3869, Z -4.6667, A 0.000, B 0.000, C 0.000 }
gfCNCPoint3[21542] = {X 82.5301, Y 47.7091, Z -4.6667, A 0.000, B 0.000, C 0.000 }
gfCNCPoint3[21543] = {X 82.0138, Y 46.8970, Z -4.6667, A 0.000, B 0.000, C 0.000 }
gfCNCPoint3[21544] = {X 81.6902, Y 45.9906, Z -4.6667, A 0.000, B 0.000, C 0.000 }
gfCNCPoint3[21545] = {X 81.5752, Y 45.0351, Z -4.6667, A 0.000, B 0.000, C 0.000 }
gfCNCPoint3[21546] = {X 81.5751, Y 44.2070, Z -4.6667, A 0.000, B 0.000, C 0.000 }
gfCNCPoint3[21547] = {X 81.6803, Y 43.2777, Z -4.6667, A 0.000, B 0.000, C 0.000 }
gfCNCPoint3[21548] = {X 81.9805, Y 42.3920, Z -4.6667, A 0.000, B 0.000, C 0.000 }
gfCNCPoint3[21549] = {X 82.4620, Y 41.5903, Z -4.6667, A 0.000, B 0.000, C 0.000 }
gfCNCPoint3[21550] = {X 83.1028, Y 40.9091, Z -4.6667, A 0.000, B 0.000, C 0.000 }
gfCNCPoint3[21551] = {X 83.1026, Y 28.5916, Z -4.6667, A 0.000, B 0.000, C 0.000 }
gfCNCPoint3[21552] = {X 79.1026, Y 28.5916, Z -4.6667, A 0.000, B 0.000, C 0.000 }
gfCNCPoint3[21553] = {X 83.1826, Y 28.5916, Z -4.6667, A 0.000, B 0.000, C 0.000 }
gfCNCPoint3[21554] = {X 83.1825, Y 16.2368, Z -4.6667, A 0.000, B 0.000, C 0.000 }
gfCNCPoint3[21555] = {X 82.5445, Y 15.5763, Z -4.6667, A 0.000, B 0.000, C 0.000 }
gfCNCPoint3[21556] = {X 82.0636, Y 14.7939, Z -4.6667, A 0.000, B 0.000, C 0.000 }
gfCNCPoint3[21557] = {X 81.7625, Y 13.9263, Z -4.6667, A 0.000, B 0.000, C 0.000 }
gfCNCPoint3[21558] = {X 81.6552, Y 13.0143, Z -4.6667, A 0.000, B 0.000, C 0.000 }
gfCNCPoint3[21559] = {X 81.6551, Y 12.1868, Z -4.6667, A 0.000, B 0.000, C 0.000 }
gfCNCPoint3[21560] = {X 81.7614, Y 11.2433, Z -4.6667, A 0.000, B 0.000, C 0.000 }
gfCNCPoint3[21561] = {X 82.0750, Y 10.3472, Z -4.6667, A 0.000, B 0.000, C 0.000 }
gfCNCPoint3[21562] = {X 82.5801, Y 9.5432, Z -4.6667, A 0.000, B 0.000, C 0.000 }
gfCNCPoint3[21563] = {X 83.2515, Y 8.8719, Z -4.6667, A 0.000, B 0.000, C 0.000 }
gfCNCPoint3[21564] = {X 84.0554, Y 8.3667, Z -4.6667, A 0.000, B 0.000, C 0.000 }
gfCNCPoint3[21565] = {X 84.9516, Y 8.0531, Z -4.6667, A 0.000, B 0.000, C 0.000 }
gfCNCPoint3[21566] = {X 85.8951, Y 7.9468, Z -4.6667, A 0.000, B 0.000, C 0.000 }
gfCNCPoint3[21567] = {X 94.0497, Y 7.9468, Z -4.6667, A 0.000, B 0.000, C 0.000 }
gfCNCPoint3[21568] = {X 94.9932, Y 8.0531, Z -4.6667, A 0.000, B 0.000, C 0.000 }
gfCNCPoint3[21569] = {X 95.8893, Y 8.3667, Z -4.6667, A 0.000, B 0.000, C 0.000 }
gfCNCPoint3[21570] = {X 96.6933, Y 8.8718, Z -4.6667, A 0.000, B 0.000, C 0.000 }
gfCNCPoint3[21571] = {X 97.3646, Y 9.5432, Z -4.6667, A 0.000, B 0.000, C 0.000 }
gfCNCPoint3[21572] = {X 97.8698, Y 10.3471, Z -4.6667, A 0.000, B 0.000, C 0.000 }
gfCNCPoint3[21573] = {X 98.1834, Y 11.2433, Z -4.6667, A 0.000, B 0.000, C 0.000 }
gfCNCPoint3[21574] = {X 98.2897, Y 12.1868, Z -4.6667, A 0.000, B 0.000, C 0.000 }
gfCNCPoint3[21575] = {X 98.2897, Y 12.9782, Z -4.6667, A 0.000, B 0.000, C 0.000 }
gfCNCPoint3[21576] = {X 98.2156, Y 13.7666, Z -4.6667, A 0.000, B 0.000, C 0.000 }
gfCNCPoint3[21577] = {X 97.9961, Y 14.5274, Z -4.6667, A 0.000, B 0.000, C 0.000 }
gfCNCPoint3[21578] = {X 97.6391, Y 15.2342, Z -4.6667, A 0.000, B 0.000, C 0.000 }
gfCNCPoint3[21579] = {X 101.8777, Y 25.7424, Z -4.6667, A 0.000, B 0.000, C 0.000 }
gfCNCPoint3[21580] = {X 101.9520, Y 25.5584, Z -4.6667, A 0.000, B 0.000, C 0.000 }
gfCNCPoint3[21581] = {X 106.1057, Y 15.2139, Z -4.6667, A 0.000, B 0.000, C 0.000 }
gfCNCPoint3[21582] = {X 105.7604, Y 14.5246, Z -4.6667, A 0.000, B 0.000, C 0.000 }
gfCNCPoint3[21583] = {X 105.5456, Y 13.7842, Z -4.6667, A 0.000, B 0.000, C 0.000 }
gfCNCPoint3[21584] = {X 105.4685, Y 13.0172, Z -4.6667, A 0.000, B 0.000, C 0.000 }
gfCNCPoint3[21585] = {X 105.4683, Y 12.1868, Z -4.6667, A 0.000, B 0.000, C 0.000 }
gfCNCPoint3[21586] = {X 105.5746, Y 11.2433, Z -4.6667, A 0.000, B 0.000, C 0.000 }
gfCNCPoint3[21587] = {X 105.8882, Y 10.3471, Z -4.6667, A 0.000, B 0.000, C 0.000 }
gfCNCPoint3[21588] = {X 106.3933, Y 9.5432, Z -4.6667, A 0.000, B 0.000, C 0.000 }
gfCNCPoint3[21589] = {X 107.0647, Y 8.8718, Z -4.6667, A 0.000, B 0.000, C 0.000 }
gfCNCPoint3[21590] = {X 107.8686, Y 8.3667, Z -4.6667, A 0.000, B 0.000, C 0.000 }
gfCNCPoint3[21591] = {X 108.7648, Y 8.0531, Z -4.6667, A 0.000, B 0.000, C 0.000 }
gfCNCPoint3[21592] = {X 109.7083, Y 7.9468, Z -4.6667, A 0.000, B 0.000, C 0.000 }
gfCNCPoint3[21593] = {X 117.7916, Y 7.9468, Z -4.6667, A 0.000, B 0.000, C 0.000 }
gfCNCPoint3[21594] = {X 118.7351, Y 8.0531, Z -4.6667, A 0.000, B 0.000, C 0.000 }
gfCNCPoint3[21595] = {X 119.6312, Y 8.3667, Z -4.6667, A 0.000, B 0.000, C 0.000 }
gfCNCPoint3[21596] = {X 120.4352, Y 8.8718, Z -4.6667, A 0.000, B 0.000, C 0.000 }
gfCNCPoint3[21597] = {X 121.1065, Y 9.5432, Z -4.6667, A 0.000, B 0.000, C 0.000 }
gfCNCPoint3[21598] = {X 121.6117, Y 10.3471, Z -4.6667, A 0.000, B 0.000, C 0.000 }
gfCNCPoint3[21599] = {X 121.9253, Y 11.2433, Z -4.6667, A 0.000, B 0.000, C 0.000 }
gfCNCPoint3[21600] = {X 122.0316, Y 12.1868, Z -4.6667, A 0.000, B 0.000, C 0.000 }
gfCNCPoint3[21601] = {X 122.0316, Y 12.9782, Z -4.6667, A 0.000, B 0.000, C 0.000 }
gfCNCPoint3[21602] = {X 121.9302, Y 13.8996, Z -4.6667, A 0.000, B 0.000, C 0.000 }
gfCNCPoint3[21603] = {X 121.6310, Y 14.7770, Z -4.6667, A 0.000, B 0.000, C 0.000 }
gfCNCPoint3[21604] = {X 121.1483, Y 15.5684, Z -4.6667, A 0.000, B 0.000, C 0.000 }
gfCNCPoint3[21605] = {X 120.5051, Y 16.2360, Z -4.6667, A 0.000, B 0.000, C 0.000 }
gfCNCPoint3[21606] = {X 120.5041, Y 40.9521, Z -4.6667, A 0.000, B 0.000, C 0.000 }
gfCNCPoint3[21607] = {X 120.5707, Y 41.0066, Z -4.6667, A 0.000, B 0.000, C 0.000 }
gfCNCPoint3[21608] = {X 121.1822, Y 41.6629, Z -4.6667, A 0.000, B 0.000, C 0.000 }
gfCNCPoint3[21609] = {X 121.6419, Y 42.4331, Z -4.6667, A 0.000, B 0.000, C 0.000 }
gfCNCPoint3[21610] = {X 121.9292, Y 43.2829, Z -4.6667, A 0.000, B 0.000, C 0.000 }
gfCNCPoint3[21611] = {X 122.0314, Y 44.1740, Z -4.6667, A 0.000, B 0.000, C 0.000 }
gfCNCPoint3[21612] = {X 122.0316, Y 45.0000, Z -4.6667, A 0.000, B 0.000, C 0.000 }
gfCNCPoint3[21613] = {X 121.9253, Y 45.9435, Z -4.6667, A 0.000, B 0.000, C 0.000 }
gfCNCPoint3[21614] = {X 121.6117, Y 46.8397, Z -4.6667, A 0.000, B 0.000, C 0.000 }
gfCNCPoint3[21615] = {X 121.1065, Y 47.6436, Z -4.6667, A 0.000, B 0.000, C 0.000 }
gfCNCPoint3[21616] = {X 120.4352, Y 48.3150, Z -4.6667, A 0.000, B 0.000, C 0.000 }
gfCNCPoint3[21617] = {X 119.6312, Y 48.8201, Z -4.6667, A 0.000, B 0.000, C 0.000 }
gfCNCPoint3[21618] = {X 118.7351, Y 49.1337, Z -4.6667, A 0.000, B 0.000, C 0.000 }
gfCNCPoint3[21619] = {X 117.7916, Y 49.2400, Z -4.6667, A 0.000, B 0.000, C 0.000 }
gfCNCPoint3[21620] = {X 111.9185, Y 49.2400, Z -4.6667, A 0.000, B 0.000, C 0.000 }
gfCNCPoint3[21621] = {X 110.9797, Y 49.1348, Z -4.6667, A 0.000, B 0.000, C 0.000 }
gfCNCPoint3[21622] = {X 110.0874, Y 48.8242, Z -4.6667, A 0.000, B 0.000, C 0.000 }
gfCNCPoint3[21623] = {X 109.2861, Y 48.3239, Z -4.6667, A 0.000, B 0.000, C 0.000 }
gfCNCPoint3[21624] = {X 108.6155, Y 47.6585, Z -4.6667, A 0.000, B 0.000, C 0.000 }
